// TwinCAT 3 PLC project Lynus_Standards
// Title: Lynus Standards
// Company: EfficientIO
// ProjectVersion: 1.0.0.2
// Description: Added FB BatteryInverter_11
// ProgramVersion: 3.1.4024.12
// libraries:
//   Tc2_EIB, * (Beckhoff Automation GmbH)
//   Tc2_MBus, * (Beckhoff Automation GmbH)
//   Tc2_Standard, * (Beckhoff Automation GmbH)
//   Tc2_SUPS, * (Beckhoff Automation GmbH)
//   Tc2_System, * (Beckhoff Automation GmbH)
//   Tc2_Utilities, * (Beckhoff Automation GmbH)
//   Tc3_BA_Common, * (Beckhoff Automation GmbH)
//   Tc3_JsonXml, * (Beckhoff Automation GmbH)
//   Tc3_Module, * (Beckhoff Automation GmbH)
// project tree:
//   Bussystems/DUTs intern/MBus Master/ ST_MBusMaster_KL6781_GVL.TcDUT
//   Bussystems/DUTs intern/RTU Master/ ST_MBRTUMaster_KL6xxx_GVL.TcDUT
//   Bussystems/ENUMs Internal/RTU Master/ E_MBRTUMaster_DeviceType.TcDUT, E_MBRTUMaster_ReadWriteMode.TcDUT
//   Bussystems/ENUMs/KNX Master/ E_Message_KNXMaster.TcDUT
//   Bussystems/ENUMs/MB RTU Master/ E_Message_MBRTUMaster.TcDUT
//   Bussystems/ENUMs/MBus Master/ E_Message_MBusMaster.TcDUT
//   Bussystems/FBs Internal/KNX Master/ FB_KNXMaster_Messages.TcPOU
//   Bussystems/FBs Internal/MBus Master/ FB_MBusMaster_Messages.TcPOU
//   Bussystems/FBs Internal/RTU Master/ FB_MBRTUMaster_Messages.TcPOU
//   Communicator/DUTs/ ST_BlockReadValue.TcDUT, ST_Content_Of_Document.TcDUT, ST_Infos_SubItem.TcDUT, ST_Message_In.TcDUT, ST_Message_Out.TcDUT, ST_SymbolRead.TcDUT, ST_Symbol_Info_SubItem.TcDUT, ST_Symbol_Upload_Info.TcDUT, ST_Symbol_Upload_Raw.TcDUT, ST_Var_Info.TcDUT, ST_Var_Info_EX.TcDUT, ST_Var_Info_EX_All.TcDUT, ST_Var_Info_GV.TcDUT, ST_Var_Info_ValueSend_GV.TcDUT, ST_Var_Info_ValueWrite_GV.TcDUT
//   Communicator/ENUMs/ eErrorMessage.TcDUT, eErrorReadWrite.TcDUT, eErrorVarInfo.TcDUT, eSavePositionFile.TcDUT, eSymbolTypeFromDocument.TcDUT
//   Communicator/FBs Internal/ FB_MessageRead.TcPOU, FB_MessageWrite.TcPOU, FB_ParsDocument.TcPOU, FB_VarInfo_ErrorCodes.TcPOU, FB_VarReadWrite_ErrorCodes.TcPOU
//   Energy/DUTs Internal/Battery Inverter/ ST_BatteryInverter_GVL.TcDUT
//   Energy/DUTs Internal/Battery/ ST_Battery_GVL.TcDUT
//   Energy/DUTs Internal/Beckhoff/ ST_KL3403.TcDUT
//   Energy/DUTs Internal/Electric CS/ ST_ECS_GVL.TcDUT
//   Energy/DUTs Internal/Electric Heating Element/ ST_EHE_GVL.TcDUT
//   Energy/DUTs Internal/Electric Meter/ ST_ElectricMeter_GVL.TcDUT
//   Energy/DUTs Internal/Generator/ ST_Generator_GVL.TcDUT
//   Energy/DUTs Internal/Grid/ ST_GridConnection_GVL.TcDUT
//   Energy/DUTs Internal/Heating Pump/ ST_HP_GVL.TcDUT
//   Energy/DUTs Internal/House/ ST_HouseConsumption_GVL.TcDUT
//   Energy/DUTs Internal/Other Big Consumer/ ST_OBC_GVL.TcDUT
//   Energy/DUTs Internal/PV/ ST_PV_GVL.TcDUT
//   Energy/DUTs Internal/System Time/ ST_Systemtime.TcDUT
//   Energy/DUTs Internal/Valve Control/ ST_Valve_Control_GVL.TcDUT
//   Energy/DUTs/Battery Inverter/ ST_BatteryInverter_Output.TcDUT
//   Energy/DUTs/Battery/ ST_Battery_Output.TcDUT
//   Energy/DUTs/Electric CS/ ST_ECS_Output.TcDUT, ST_Setup_ECS.TcDUT
//   Energy/DUTs/Electric Heating Element/ ST_EHE_Output.TcDUT, ST_Setup_EHE.TcDUT
//   Energy/DUTs/Electric Meter/ ST_ElectricMeter_Output_Power.TcDUT, ST_ElectricMeter_Output_Counter.TcDUT
//   Energy/DUTs/Generator/ ST_Generator_Output.TcDUT, ST_Setup_Generator.TcDUT
//   Energy/DUTs/Grid/ ST_GridConnection_Output.TcDUT
//   Energy/DUTs/Heating pump/ ST_HP_Output.TcDUT, ST_Setup_HP.TcDUT
//   Energy/DUTs/House/ ST_HouseConsumption_Output.TcDUT
//   Energy/DUTs/Other Big Consumer/ ST_OBC_Output.TcDUT, ST_Setup_OBC.TcDUT
//   Energy/DUTs/PV/ ST_PV_Output.TcDUT
//   Energy/DUTs/Temperature/ ST_InputData_KL320x.TcDUT, ST_OutputData_KL320x.TcDUT, ST_Temperature_Output.TcDUT
//   Energy/DUTs/Valve Control/ ST_Valve_Control_Output.TcDUT
//   Energy/ENUMs Internal/Temperature/ E_ChooseSensortype_KL320x.TcDUT, E_Step_Config_Terminal_KL320x.TcDUT
//   Energy/ENUMs/Battery Inverter/ E_Message_BatteryInverter.TcDUT
//   Energy/ENUMs/Battery/ E_Message_Battery.TcDUT
//   Energy/ENUMs/Electric Charging Station/ E_Message_ECS.TcDUT
//   Energy/ENUMs/Electric Heating Element/ E_Message_EHE.TcDUT
//   Energy/ENUMs/Electric Meter/ E_Message_EM.TcDUT
//   Energy/ENUMs/EMS/ E_Message_EMS.TcDUT
//   Energy/ENUMs/Generator/ E_Message_Generator.TcDUT
//   Energy/ENUMs/Grid/ E_Message_Grid.TcDUT
//   Energy/ENUMs/Heating Pump/ E_Message_HP.TcDUT
//   Energy/ENUMs/House Consumption/ E_Message_HouseC.TcDUT
//   Energy/ENUMs/Other Big Consumer/ E_Message_OBC.TcDUT
//   Energy/ENUMs/PV/ E_Message_PV.TcDUT
//   Energy/ENUMs/Temperature/ E_Message_Temperature.TcDUT
//   Energy/ENUMs/Valve Control/ E_Message_ValveControl.TcDUT
//   Energy/FBs Internal/Battery Inverter/ FB_BatteryInverter.TcPOU, FB_BatteryInverter_11.TcPOU
//   Energy/FBs Internal/Battery/ FB_Battery.TcPOU
//   Energy/FBs Internal/Beckhoff/ FB_KL3403_SimpleProcessImage.TcPOU, FB_XL1XXX_DI.TcPOU, FB_XL2XXX_DO.TcPOU, FB_XL3XXX_AI.TcPOU, FB_XL4XXX_AO.TcPOU
//   Energy/FBs Internal/Controller/ FB_PID.TcPOU
//   Energy/FBs Internal/Electric CS/ FB_ElectricChargingStation.TcPOU
//   Energy/FBs Internal/Electric Heating Element/ FB_ElectricHeatingElement.TcPOU
//   Energy/FBs Internal/Electric Meter/ FB_ElectricMeter.TcPOU
//   Energy/FBs Internal/EMS/ FB_EMS_Message.TcPOU
//   Energy/FBs Internal/Energy Counter/ FB_EnergyCounter.TcPOU
//   Energy/FBs Internal/Generator/ FB_Generator.TcPOU
//   Energy/FBs Internal/Grid/ FB_GridConnection.TcPOU
//   Energy/FBs Internal/Heating Pump/ FB_HeatingPump.TcPOU
//   Energy/FBs Internal/House/ FB_HouseConsumption.TcPOU
//   Energy/FBs Internal/Other Big Consumer/ FB_BigConsumer.TcPOU
//   Energy/FBs Internal/PV/ FB_PV_Production.TcPOU
//   Energy/FBs Internal/Valve Control/ FB_Valve_Control.TcPOU
//   General/DUTs Internal/Convert/ eByteOrder.TcDUT, ST_UN_FLOAT_CONVERT_DWORD_REAL.TcDUT, ST_UN_FLOAT_CONVERT_ULINT_LREAL.TcDUT
//   General/DUTs Internal/Devices/ ST_NumberOfDevices_GVL.TcDUT
//   General/FBs Internal/Convert/BOOL/ FB_CV_BOOL_TO_WORD.TcPOU, FB_CV_WORD_TO_BOOL.TcPOU
//   General/FBs Internal/Convert/BYTE/ FB_CV_BYTE_TO_WORD.TcPOU, FB_CV_WORD_TO_BYTE.TcPOU
//   General/FBs Internal/Convert/DINT/ FB_CV_DINT_TO_WORD.TcPOU, FB_CV_WORD_TO_DINT.TcPOU
//   General/FBs Internal/Convert/DWORD/ FB_CV_DWORD_TO_WORD.TcPOU, FB_CV_WORD_TO_DWORD.TcPOU
//   General/FBs Internal/Convert/INT/ FB_CV_INT_TO_WORD.TcPOU, FB_CV_WORD_TO_INT.TcPOU
//   General/FBs Internal/Convert/LINT/ FB_CV_LINT_TO_WORD.TcPOU, FB_CV_WORD_TO_LINT.TcPOU
//   General/FBs Internal/Convert/LREAL_FLOAT/ FB_CV_LREAL_FLOAT_TO_WORD.TcPOU, FB_CV_WORD_TO_LREAL_FLOAT.TcPOU
//   General/FBs Internal/Convert/LWORD/ FB_CV_LWORD_TO_WORD.TcPOU, FB_CV_WORD_TO_LWORD.TcPOU
//   General/FBs Internal/Convert/REAL_FLOAT/ FB_CV_REAL_FLOAT_TO_WORD.TcPOU, FB_CV_WORD_TO_REAL_FLOAT.TcPOU
//   General/FBs Internal/Convert/SINT/ FB_CV_SINT_TO_WORD.TcPOU, FB_CV_WORD_TO_SINT.TcPOU
//   General/FBs Internal/Convert/UDINT/ FB_CV_UDINT_TO_WORD.TcPOU, FB_CV_WORD_TO_UDINT.TcPOU
//   General/FBs Internal/Convert/ULINT/ FB_CV_ULINT_TO_WORD.TcPOU, FB_CV_WORD_TO_ULINT.TcPOU
//   General/FBs Internal/Convert/USINT/ FB_CV_USINT_TO_WORD.TcPOU, FB_CV_WORD_TO_USINT.TcPOU
//   General/FBs Internal/Filter/ FB_Filter.TcPOU
//   General/FBs Internal/Linear Interpolation/ FB_Lin_Interpolation.TcPOU
//   General/FBs Internal/Number Of Device/ FB_NumberOfDevice.TcPOU
//   General/FUNs Internal/ ARRAY_AVG.TcPOU, F_Scalvalue.TcPOU
//   GVL and CONST/Bussystems/ Constants_Bussystems.TcGVL, GVL_Bussystems.TcGVL
//   GVL and CONST/Energy/ Constants_Energy.TcGVL, GVL_Energy.TcGVL
//   GVL and CONST/Communicator/ GVL_Communicator.TcGVL, Constants_Communicator.TcGVL
//   GVL and CONST/General/ Constants_General.TcGVL
//   GVL and CONST/Persistent Data/ GVL_Persistent_Data.TcGVL
//   GVL and CONST/Sensors/ Constants_Sensors.TcGVL, GVL_Sensors.TcGVL
//   Persistent Data/FBs Internal/PD Slave/ FB_PersistentData_Number.TcPOU, FB_PersistentData_String.TcPOU
//   Sensors/DUTs Internal/Temperature/ ST_Temperature_GVL.TcDUT
//   Sensors/FBs Internal/Temperature/ FB_Config_KL320x.TcPOU, FB_TempSensor_M50_P200.TcPOU

// ---- Bussystems/DUTs intern/MBus Master/ST_MBusMaster_KL6781_GVL.TcDUT
{attribute 'conditionalshow'}
TYPE ST_MBusMaster_KL6781_GVL :
STRUCT
	{attribute 'hide'}
	stDataMBusCommunicationKL6781					: ST_MBus_Communication;					//Datastrcut between the KL6781 and the other Functionblocks
	{attribute 'hide'}			
	eBaudrateMBusKL6781								: E_MBus_Baudrate;							//With this Baudrate the Functionsblocks for the Counters are reading out
END_STRUCT
END_TYPE

// ---- Bussystems/DUTs intern/RTU Master/ST_MBRTUMaster_KL6xxx_GVL.TcDUT
{attribute 'conditionalshow'}
TYPE ST_MBRTUMaster_KL6xxx_GVL :
STRUCT
	{attribute 'hide'}
	bSlaveStartReadOrWrite				: BOOL;																		//RTU Slave send to the RTU Master the start for read or write command
	{attribute 'hide'}
	bTerminalIsConfigured				: BOOL;																		//The RTU Master set this Flag to True when the Terminal is successfully configured
	{attribute 'hide'}	
	bReadWriteIsDone					: BOOL;																		//The Slave Set this to True when all Registers are done. (For Eg. in the Last Step of the Statemachine) The Master Reset this Flag. So then next Modbus Adress can be processed.
	{attribute 'hide'}
	bMasterIsBusy						: BOOL;																		//RTU Master is busy. 
	{attribute 'hide'}
	bNoNewMBusAdress					: BOOL;																		//When this Flag is true, the Client Functions not can set a new Modbus Slave Adress
	{attribute 'hide'}
	byErrorWarning						: BYTE;																		//Error Warning State
	{attribute 'hide'}
	byActualMBAdressInProgrss			: BYTE;																		//Actual Modbus Slave Adress what is in Progress at the moment
	{attribute 'hide'}
	byNumberOfSlaves					: BYTE;																		//Number of Slaves on several Line
	{attribute 'hide'}
	wModbusRegister						: WORD;																		//The Modbus Register from the Slave for the Master to read/write
	{attribute 'hide'}	
	wNumberOfRegister					: WORD;																		//Number of Registers from the Slave to the Master for read/write 
	{attribute 'hide'}
	arrAllModbusSlaveAdresses			: ARRAY[1..247] OF BYTE;													//Array with all Modbuis Slave Adresses				
	{attribute 'hide'}
	arrReadOutData						: ARRAY[1..Constants_Bussystems.wQuantityOfRegistersMBRTUMaster] OF WORD;	//Data after Reading to send from the Master to the Slave
	{attribute 'hide'}
	arrWriteOutData						: ARRAY[1..Constants_Bussystems.wQuantityOfRegistersMBRTUMaster] OF WORD;	//Data to send from the Save to the Master for writing
	{attribute 'hide'}
	eMBRTUReadWriteMode					: E_MBRTUMaster_ReadWriteMode;												//Choose between the different Modbus Actions
	{attribute 'hide'}
	eMBRTUDeviceType					: E_MBRTUMaster_DeviceType;													//The Slave send to the Master the Device Type. Only the same Device Types are Allowed on 1 Backhoff Terminal
END_STRUCT
END_TYPE

// ---- Bussystems/ENUMs Internal/RTU Master/E_MBRTUMaster_DeviceType.TcDUT
{attribute 'qualified_only'}
{attribute 'strict'}
{attribute 'conditionalshow'}
TYPE E_MBRTUMaster_DeviceType :
(
	//Device Types on the RTU Bus, to configure the Terminal
	{attribute 'hide'}
	eNoModbusRTUDevice								:= 0,
	{attribute 'hide'}
	ePilotPMAC201_HW								:= 1,
	{attribute 'hide'}				
	eDrexelAWeiss_AereosilentStratosLU_Ventilation	:= 2,
	{attribute 'hide'}
	eABB_CM_UFD_M31M_NAProtection					:= 3,
	{attribute 'hide'}
	eSchrack_ECS_CIONHOME_SEMIPUBLIC				:= 4,
	{attribute 'hide'}
	ePV_DeltaSunspec								:= 5
);
END_TYPE

// ---- Bussystems/ENUMs Internal/RTU Master/E_MBRTUMaster_ReadWriteMode.TcDUT
{attribute 'qualified_only'}
{attribute 'strict'}
{attribute 'conditionalshow'}
TYPE E_MBRTUMaster_ReadWriteMode :
(
	{attribute 'hide'}
	eModbusRTUMaster_NoMode := 0,
	{attribute 'hide'}
	eModbusRTUMaster_ReadCoils	:= 1,									//Read binary Outputs
	{attribute 'hide'}
	eModbusRTUMaster_ReadInputStatus	:= 2,							//Read binary Inputs
	{attribute 'hide'}
	eModbusRTUMaster_ReadRegs	:= 3,									//Read Output Registers
	{attribute 'hide'}
	eModbusRTUMaster_ReadInputRegs	:= 4,								//Read Input Registers
	{attribute 'hide'}
	eModbusRTUMaster_WriteSingleCoil	:= 5,							//Write 1 binary Outputs
	{attribute 'hide'}
	eModbusRTUMaster_WriteSingleRegister	:= 6,						//Write a single Register
	{attribute 'hide'}
	eModbusRTUMaster_Diagnostics	:= 8,								//Send a Diagnostic request
	{attribute 'hide'}
	eModbusRTUMaster_WriteMultipleCoils	:= 15,							//Write more binary Outputs 
	{attribute 'hide'}
	eModbusRTUMaster_WriteRegs	:= 16									//Write more then one Register
);
END_TYPE

// ---- Bussystems/ENUMs/KNX Master/E_Message_KNXMaster.TcDUT
{attribute 'qualified_only'}
{attribute 'strict'}
TYPE E_Message_KNXMaster :
(
	eAllOk := 0,
	eTooMuchKNXMasters := 1,
	eNoConnectionToBackend := 2,
	eWrong_KNX_Phys_Addr := 3,
	eWrong_KNX_Group_Addr := 4,
	eWrong_KNX_Group_Len := 5,
	eWrong_KNX_No_Filter := 6,
	eWrong_KNX_Firmware := 7,
	eWrong_KNX_Mode := 8,
	eWrong_Mode := 9,
	eWrong_KNX_Firmware_B1_Necessary := 10,
	eWrong_KNX_Firmware_B3_Necessary := 11,
	eWrong_KNX_Data_Len := 12,
	eError_KNX_Service_Not_Support := 13,
	eKL6301_TP_Toggle_Error := 14,
	eTime_Out := 15,
	eKL6301_No_Response_from_Terminal := 16,
	eError_Send_8Bit_Wrong_Scaling_Mode := 17,
	eError_KNX_Phy_Addr_Not_Support := 18,
	eError_KNX_Write_Data := 19,
	eMonitor_Mode_Len_Is_Not_Ok_Must_0 := 20,
	eMonitor_Mode_Addr_Is_Not_Ok_Must_0 := 21,
	eWatchdog_Error_No_Send := 22,
	eError_KNX_No_Ack := 23,
	eError_KNX_No_Com_To_TP := 24,
	eError_TP_Temp_Warning := 25,
	eError_TP_Protocol_Error := 26,
	eError_TP_Transmitter_Error := 27,
	eError_TP_Receive_Error := 28,
	eError_TP_Slave_Collision := 29
);
END_TYPE

// ---- Bussystems/ENUMs/MB RTU Master/E_Message_MBRTUMaster.TcDUT
{attribute 'qualified_only'}
{attribute 'strict'}
TYPE E_Message_MBRTUMaster :
(
	eAllOk := 0,
	eNoTerminalConfiguration := 1,
	eTooMuchMBRTUMasters := 2,
	eNoConnectionToBackend := 3,
	eTerminalConfigurationError := 4,
	eModbusErrorIllegalFunction := 5,
	eModbusErrorIllegalDataAdress := 6,
	eModbusErrorIllegalDataValue := 7,
	eModbusErrorSlaveDeviceFailure := 8,
	eModbusErrorAcknowledge := 9,
	eModbusErrorSlaveDeviceBusy := 10,
	eModbusErrorNegativeAcknowledge := 11,
	eModbusErrorMemoryParity := 12,
	eModbusErrorGatewayPathUnavailable := 13,
	eModbusErrorGatewayTargetDeviceFailedToRespond := 14,
	eModbusErrorCharrecTimeout := 15,
	eModbusErrorIllegalDataSize := 16,
	eModbusErrorIllegalDeviceAdress := 17,
	eModbusErrorIllegalDestinationAdress := 18,
	eModbusErrorIllegalDestinationSize := 19,
	eModbusErrorNoResponse := 20,
	eModbusErrorTxBufferOverrun := 21,
	eModbusErrorSendTimeout := 22,
	eModbusErrorDataSizeOverrun := 23,
	eModbusErrorStringOverrun := 24,
	eModbusErrorInvalidPointer := 25,
	eModbusErrorCRC := 26,
	eModbusErrorInvalidMemoryAdress := 27,
	eModbusErrorTransmitBufferTooSmal := 28
);
END_TYPE

// ---- Bussystems/ENUMs/MBus Master/E_Message_MBusMaster.TcDUT
{attribute 'qualified_only'}
{attribute 'strict'}
TYPE E_Message_MBusMaster :
(
	eAllOk := 0,
	eTooMuchMBusMasters := 1,
	eNoConnectionToBackend := 2,
	eMBUSERROR_CIField_wrong_72hex_expected  := 3,
 	eMBUSERROR_no_data_received := 4,
  	eMBUSERROR_error_checksum := 5,
  	eMBUSERROR_error_in_head_data := 6,
 	eMBUSERROR_usiAddress_over_250 := 7,
  	eMBUSERROR_send_error := 8,
  	eMBUSERROR_received_address_wrong := 9,
  	eMBUSERROR_cMBUS_MaxCom_below_1 := 10,
  	eMBUSERROR_iComId_over_cMBUS_MaxCom := 11,
  	eMBUSERROR_manufacturer_sign_wrong := 12,
  	eMBUSERROR_baudrate_wrong := 13,
  	eMBUSERROR_ReceiveBufferFull := 14,
  	eMBUSERROR_E5hex_no_received := 15,
  	eMBUSERROR_no_stop_character := 16,
  	eMBUSERROR_length_wrong := 17,
  	eMBUSERROR_wrong_terminal := 18,
  	eMBUSERROR_Terminal_is_not_initialized := 19,
  	eMBUSERROR_stSecAdr_udiIdNumber_wrong := 20,
  	eMBUSERROR_missing_parts_telegram := 21,
  	eMBUSERROR_no_stop_character_received := 22,
  	eMBUSERROR_too_many_characters := 23,
  	eMBUSERROR_TimeOut_FB_KL6781 := 24,
  	eMBUSERROR_TimeOut_MeterFB := 25,
	eMBUSERROR_COM_PARAMETERCHANGED := 26,
  	eMBUSERROR_COM_TXBUFFOVERRUN := 27,
  	eMBUSERROR_COM_STRINGOVERRUN := 28,
  	eMBUSERROR_COM_ZEROCHARINVALID := 29,
  	eMBUSERROR_COM_INVALIDPOINTER := 30,
 	eMBUSERROR_COM_INVALIDRXPOINTER := 31,
  	eMBUSERROR_COM_INVALIDRXLENGTH := 32,
  	eMBUSERROR_COM_DATASIZEOVERRUN := 33,
  	eMBUSERROR_COM_INVALIDBAUDRATE := 34,
  	eMBUSERROR_COM_INVALIDNUMDATABITS := 35,
  	eMBUSERROR_COM_INVALIDNUMSTOPBITS := 36,
  	eMBUSERROR_COM_INVALIDPARITY := 37,
  	eMBUSERROR_COM_INVALIDHANDSHAKE := 38,
  	eMBUSERROR_COM_INVALIDNUMREGISTERS := 39,
  	eMBUSERROR_COM_INVALIDREGISTER := 40,
  	eMBUSERROR_COM_TIMEOUT := 41
);
END_TYPE

// ---- Communicator/DUTs/ST_BlockReadValue.TcDUT
{attribute 'conditionalshow'}
TYPE ST_BlockReadValue :
STRUCT
	{attribute 'hide'}
	udiIndexGroup			: UDINT;						//Index group from symbol  
	{attribute 'hide'}
	udiIndexOffset			: UDINT;						//Index offset from symbol
	{attribute 'hide'}
	udiLength				: UDINT;						//Index length from symbol
END_STRUCT
END_TYPE

// ---- Communicator/DUTs/ST_Content_Of_Document.TcDUT
{attribute 'conditionalshow'}
TYPE ST_Content_Of_Document :
STRUCT
	{attribute 'hide'}
	sSymbolName				: STRING(48);																				//Symbol Name
	{attribute 'hide'}
	eSymbolType				: eSymbolTypeFromDocument;																	//Symbol Type (Enum, Struct or FB)
	{attribute 'hide'}
	arrSubItemName			: ARRAY[1..Constants_Communicator.uiArraySizeOfMarkedSubItems] OF STRING(48);				//Name from the Subitems
	{attribute 'hide'}
	arrSubItemSymbolType	: ARRAY[1..Constants_Communicator.uiArraySizeOfMarkedSubItems] OF STRING(255);				//Type from the Subitems
	{attribute 'hide'}
	arrSubItemUnit			: ARRAY[1..Constants_Communicator.uiArraySizeOfMarkedSubItems] OF STRING(255);				//Unit from the SubItem
	{attribute 'hide'}
	arrSubItemTextEnum		: ARRAY[1..Constants_Communicator.uiArraySizeOfMarkedSubItems] OF STRING(48);				//Text from Enum
	{attribute 'hide'}
	arrSubItemIndexEnum		: ARRAY[1..Constants_Communicator.uiArraySizeOfMarkedSubItems] OF STRING(6);				//Index-Value from Enum
END_STRUCT
END_TYPE

// ---- Communicator/DUTs/ST_Infos_SubItem.TcDUT
{attribute 'conditionalshow'}
TYPE ST_Infos_SubItem :
STRUCT
	{attribute 'hide'}
	bIsEnum						: BOOL;						//Is true if the symbol is a enum		
	{attribute 'hide'}				
	sSubItemName				: STRING(48);				//Name of the Sub Item	
	{attribute 'hide'}								
	sSubItemType				: STRING(255);				//Type of the sub item
	{attribute 'hide'}									
	sSubItemUnit				: STRING(255);				//Unit of the sub item
	{attribute 'hide'}									
	uiSizeArray					: UINT;						//Array size if symbol type is a array
	{attribute 'hide'}
	udiSubItemGroup				: UDINT;					//Group number of sub item
	{attribute 'hide'}
	udiSubItemOffset			: UDINT;					//Offset of group number of sub item
	{attribute 'hide'}
	udiSubItemSize				: UDINT;					//Size of sub item variable in Byte 
END_STRUCT
END_TYPE

// ---- Communicator/DUTs/ST_Message_In.TcDUT
{attribute 'conditionalshow'}
TYPE ST_Message_In :
STRUCT
	{attribute 'hide'}
	sFullSymbolName				: STRING(48);															//Full Symbol name of plc variable uncoded
	{attribute 'hide'}
	sSymbolUnit					: STRING(255);															//Symbol unit of plc variable uncoded
	{attribute 'hide'}
	sSymbolType					: STRING(255);															//Symbol type of plc variable uncoded	
	{attribute 'hide'}
	arrValue					: ARRAY[1..Constants_Communicator.bySizeOfValueArray] OF STRING(30);	//Value from the Variable	
END_STRUCT
END_TYPE

// ---- Communicator/DUTs/ST_Message_Out.TcDUT
{attribute 'conditionalshow'}
TYPE ST_Message_Out :
STRUCT
	{attribute 'hide'}
	sFullSymbolName				: STRING(48);																			//Symbol name of plc variable uncoded
	{attribute 'hide'}
	sSymbolType					: STRING(255);																			//Symbol type of plc variable uncoded
	{attribute 'hide'}
	uiSizeArray					: UINT;																					//Size of actuall Array
	{attribute 'hide'}
	byReadWriteArrayNumber		: BYTE;																					//Number of the array for which the command is intended
	{attribute 'hide'}
	arrValue					: ARRAY[0..Constants_Communicator.bySizeOfReceivedValueArrayInJson] OF STRING(30);		//Value from the Variable	
END_STRUCT
END_TYPE

// ---- Communicator/DUTs/ST_SymbolRead.TcDUT
{attribute 'conditionalshow'}
TYPE ST_SymbolRead :
STRUCT
	{attribute 'hide'}
	sFullSymbolName				: STRING(48);																	//Full Symbol name of plc variable uncoded
	{attribute 'hide'}
	arrValue					: ARRAY[1..Constants_Communicator.bySizeOfValueArray] OF STRING(30);			//Value from the Variable	
END_STRUCT
END_TYPE

// ---- Communicator/DUTs/ST_Symbol_Info_SubItem.TcDUT
{attribute 'conditionalshow'}
TYPE ST_Symbol_Info_SubItem :
STRUCT
	{attribute 'hide'}
	udiSubItemGroup				: UDINT;					//Group number of sub item
	{attribute 'hide'}
	udiSubItemOffset			: UDINT;					//Offset of group number of sub item
	{attribute 'hide'}
	udiSubItemSize				: UDINT;					//Size of sub item variable in Byte
END_STRUCT
END_TYPE

// ---- Communicator/DUTs/ST_Symbol_Upload_Info.TcDUT
{attribute 'conditionalshow'}
TYPE ST_Symbol_Upload_Info :
STRUCT
	{attribute 'hide'}
	udiSymbols				: UDINT;				//Number of symbols on plc
	{attribute 'hide'}
	udiSymbolSize			: UDINT;				//Size of symbols on plc
END_STRUCT
END_TYPE

// ---- Communicator/DUTs/ST_Symbol_Upload_Raw.TcDUT
{attribute 'conditionalshow'}
TYPE ST_Symbol_Upload_Raw :
STRUCT
	{attribute 'hide'}
	udiSymbolName				: UDINT;				//Symbol name of plc variable in coded format
	{attribute 'hide'}
	udiGroup					: UDINT;				//Group number
	{attribute 'hide'}
	udiOffset					: UDINT;				//Offset of group number
	{attribute 'hide'}
	udiSize						: UDINT;				//Size of variable
	{attribute 'hide'}
	udiAdsDataType				: UDINT;				//Ads Data Type
	{attribute 'hide'}
	udiFlags					: UDINT;				//Flags
	{attribute 'hide'}
	uiNameLength				: UINT;					//Length of the symbol name
	{attribute 'hide'}
	uiTypeLength				: UINT;					//Lenght of the type in Byte it is bigdata ads type
	{attribute 'hide'}
	uiCommentLength				: UINT;					//Comment lenght
END_STRUCT
END_TYPE

// ---- Communicator/DUTs/ST_Var_Info.TcDUT
{attribute 'conditionalshow'}
TYPE ST_Var_Info :
STRUCT
	{attribute 'hide'}
	sSymbolName					: STRING(255);			//Symbol name of plc variable uncoded
	{attribute 'hide'}
	uiSizeArray					: UINT;					//Array size if symbol type is a array
	{attribute 'hide'}
	udiGroup					: UDINT;				//Group number
	{attribute 'hide'}
	udiOffset					: UDINT;				//Offset of group number
	{attribute 'hide'}
	udiSize						: UDINT;				//Size of variable
	{attribute 'hide'}
	udiFlags					: UDINT;				//Flags
	{attribute 'hide'}
	uiTypeLength				: UINT;					//Lenght of the type in Byte it is bigdata ads type
	{attribute 'hide'}
	sAdsDataType				: STRING(12);			//ADS data type	
	{attribute 'hide'}
	sSymbolType					: STRING(255);			//Symbol type of plc variable uncoded
	{attribute 'hide'}
	sSymbolComment				: STRING(255);			//Symbol comment of plc variable uncoded
END_STRUCT
END_TYPE

// ---- Communicator/DUTs/ST_Var_Info_EX.TcDUT
{attribute 'conditionalshow'}
TYPE ST_Var_Info_EX :
STRUCT
	{attribute 'hide'}
	bNoStandardDatatypeDetected	: BOOL;																					//If its true the Symbol is not a standart Data Type			
	{attribute 'hide'}
	sFullSymbolName				: STRING(48);																			//Full Symbol name of plc variable 
	{attribute 'hide'}
	sSymbolName					: STRING(255);																			//Symbol name of plc variable 
	{attribute 'hide'}
	uiSizeArray					: UINT;																					//Array size if symbol type is a array
	{attribute 'hide'}
	udiGroup					: UDINT;																				//Group number
	{attribute 'hide'}
	udiOffset					: UDINT;																				//Offset of group number
	{attribute 'hide'}
	udiSize						: UDINT;																				//Size of variable in Byte	
	{attribute 'hide'}
	uiTypeLength				: UINT;																					//Lenght of the type in Byte it is bigdata ads type
	{attribute 'hide'}
	udiFlags					: UDINT;																				//Flags
	{attribute 'hide'}
	sAdsDataType				: STRING(12);																			//ADS data type	
	{attribute 'hide'}
	sSymbolType					: STRING(255);																			//Symbol type of plc variable	
	{attribute 'hide'}
	sSymbolUnit					: STRING(255);																			//Symbol Unit
	{attribute 'hide'}
	sProjectName				: STRING(63);																			//Projekt Name			
	{attribute 'hide'}
	arrInfoSubItems				: ARRAY[1..Constants_Communicator.uiArraySizeOfMarkedSubItems] OF ST_Infos_SubItem; 	//All important infos from the SubItems it is not a standart Data Type
END_STRUCT
END_TYPE

// ---- Communicator/DUTs/ST_Var_Info_EX_All.TcDUT
{attribute 'conditionalshow'}
TYPE ST_Var_Info_EX_All :
STRUCT
	{attribute 'hide'}
	sFullSymbolName				: STRING(48);			//Full Symbol name of plc variable
	{attribute 'hide'}
	uiSizeArray					: UINT;					//Array size if symbol type is a array
	{attribute 'hide'}
	udiGroup					: UDINT;				//Group number
	{attribute 'hide'}
	udiOffset					: UDINT;				//Offset of group number
	{attribute 'hide'}
	udiSize						: UDINT;				//Size of variable in Byte	
	{attribute 'hide'}
	sSymbolType					: STRING(255);			//Symbol Type
	{attribute 'hide'}
	sSymbolUnit					: STRING(255);			//Comment from the symbol
END_STRUCT
END_TYPE

// ---- Communicator/DUTs/ST_Var_Info_GV.TcDUT
{attribute 'conditionalshow'}
TYPE ST_Var_Info_GV :
STRUCT
	{attribute 'hide'}
	sFullSymbolName				: STRING(48);			//Full Symbol name of plc variable uncoded
	{attribute 'hide'}
	uiSizeArray					: UINT;					//Array size if symbol type is a array
	{attribute 'hide'}
	udiGroup					: UDINT;				//Group number
	{attribute 'hide'}
	udiOffset					: UDINT;				//Offset of group number
	{attribute 'hide'}
	udiSize						: UDINT;				//Size of variable in Byte	
	{attribute 'hide'}
	sSymbolType					: STRING(255);			//Symbol Type
	{attribute 'hide'}
	sSymbolUnit					: STRING(255);			//Comment from the symbol	
END_STRUCT
END_TYPE

// ---- Communicator/DUTs/ST_Var_Info_ValueSend_GV.TcDUT
{attribute 'conditionalshow'}
TYPE ST_Var_Info_ValueSend_GV :
STRUCT
	//Values from ads read function
	{attribute 'hide'}
	sFullSymbolName				: STRING(48);																	//Full Symbol name of plc variable uncoded
	{attribute 'hide'}
	sSymbolType					: STRING(255);																	//Symbol type of plc variable uncoded	
	{attribute 'hide'}
	sSymbolUnit					: STRING(255);																	//Symbol Unit
	{attribute 'hide'}
	arrValue					: ARRAY[1..Constants_Communicator.bySizeOfValueArray] OF STRING(30);			//Value from the Variable
	//Values from sending function and buffer
	{attribute 'hide'}
	bBufferOK					: BOOL;																			//Buffer state ok
	{attribute 'hide'}
	bBusy						: BOOL;																			//Send Message is busy
	{attribute 'hide'}
	bErrorSending				: BOOL;																			//After send messege success a error	
	{attribute 'hide'}
	udiCountBuffer				: UDINT;																		//Return the counter of stored values in the buffer after read	
END_STRUCT
END_TYPE

// ---- Communicator/DUTs/ST_Var_Info_ValueWrite_GV.TcDUT
{attribute 'conditionalshow'}
TYPE ST_Var_Info_ValueWrite_GV :
STRUCT
	//Received from external to ads write function
	{attribute 'hide'}
	bWriteNewValue				: BOOL;																			//New Value received to write
	{attribute 'hide'}
	bSendFunctionOK				: BOOL;																			//Necessary to start read/write
	{attribute 'hide'}
	uiSizeArray					: UINT;																			//Size of actuall Array
	{attribute 'hide'}
	udiCountBuffer				: UDINT;																		//Return the counter of stored values in the reveived buffer
	{attribute 'hide'}
	sFullSymbolName				: STRING(48);																	//Full Symbol name of plc variable uncoded
	{attribute 'hide'}
	sSymbolType					: STRING(255);																	//Symbol type of plc variable uncoded	
	{attribute 'hide'}
	arrValue					: ARRAY[1..Constants_Communicator.bySizeOfValueArray] OF STRING(30);			//Value from the Variable
	//State from ads write function to received function buffer
	{attribute 'hide'}
	bBusy						: BOOL;																			//Write Message is busy
	{attribute 'hide'}
	bErrorWrite					: BOOL;																			//After write the messege success a error		
END_STRUCT
END_TYPE

// ---- Communicator/ENUMs/eErrorMessage.TcDUT
{attribute 'qualified_only'}
{attribute 'strict'}
TYPE eErrorMessage :
(
	eNoError							:= 0,
	eReceivedMessageWithError			:= 1,
	eReceivedMessageIncompatibility		:= 2,
	eCreatedMessageWithError			:= 3
);
END_TYPE

// ---- Communicator/ENUMs/eErrorReadWrite.TcDUT
{attribute 'qualified_only'}
{attribute 'strict'}
TYPE eErrorReadWrite :
(
	eNoError							:= 0,
	eErrorRead							:= 1,
	eErrorWrite							:= 2,
	eErrorSizeFloatValueRead			:= 3,
	eErrorSizeValueWrite				:= 4
);
END_TYPE

// ---- Communicator/ENUMs/eErrorVarInfo.TcDUT
{attribute 'qualified_only'}
{attribute 'strict'}
TYPE eErrorVarInfo :
(
	eNoError								:= 0,
	eArraySizeError							:= 1,
	eTimoutError							:= 2,
	eCommentLenghtError						:= 3,
	eCommentDescriptionError				:= 4,
	eSymbolTypeError						:= 5,
	eSymbolNameToLongError					:= 6,
	eReadWriteFunctionToMuch				:= 7,
	eVarInfoFunctionToMuch					:= 8,
	eSendReceiveFunctionToMuch				:= 9,
	eMoreReadWriteFuctionsAsSymbols			:= 10,
	eNoTMCFileSelected						:= 11,
	eArrayWithNoStandartDatatype			:= 12,
	eSymbolNotFoundInTMCFile				:= 13,
	eSymbolNameWithSubItemIsToLong			:= 14,
	eToMuchSubItemsInSymbol					:= 15,
	eToMuchSymbols							:= 16,
	eSubItemsInfoError						:= 17,
	eNoSendReceiveFunction					:= 18,
	eNoReadWriteFunction					:= 19,
	eNoSymbolsFound							:= 20,
	eTMCFileTimoutError						:= 100,
	eTMCFileContentOfSymbolIsToBig			:= 101,
	eTMCFileSymbolNameToLongError			:= 102,
	eTMCFileToMuchSubItemsInOneSymbol		:= 103,
	eTMCFileSubItemNameToLongError			:= 104,
	eTMCFileErrorWhenOpeningTheFile			:= 105,
	eTMCFileErrorWhenReadingTheFile			:= 106,
	eTMCFileErrorWhenClosingTheFile			:= 107,
	eTMCFileToMuchNoStandartDatatypes		:= 108,
	eTMCFileEnumNameToLongError				:= 109,
	eTMCFileEnumIndexToMuchSizes			:= 110,
	eTMCFileArraySizeError					:= 111,
	eTMCFileStringSizeError					:= 112,
	eTMCFileCheckPositionError				:= 113,
	eTMCFileSearchPositionError				:= 114,
	eTMCFileMissingSubItems					:= 115,
	eTMCFileFunctionblockAccessNotAllowed	:= 116,
	eTMCFileToMuchSubItemsInOtherSubItems	:= 117,
	eTMCFileArrayWithNoStandartDatatype		:= 118
);
END_TYPE

// ---- Communicator/ENUMs/eSavePositionFile.TcDUT
{attribute 'qualified_only'}
{attribute 'strict'}
{attribute 'conditionalshow'}
TYPE eSavePositionFile :
(
	{attribute 'hide'}
	ePostionHardDisk := 0,
	{attribute 'hide'}
	ePostionC := 1
);
END_TYPE

// ---- Communicator/ENUMs/eSymbolTypeFromDocument.TcDUT
{attribute 'qualified_only'}
{attribute 'strict'}
{attribute 'conditionalshow'}
TYPE eSymbolTypeFromDocument :
(
	{attribute 'hide'}
	eNoInformation		:= 0,
	{attribute 'hide'}
	eIsEnum				:= 1,
	{attribute 'hide'}
	eIsStruct			:= 2,
	{attribute 'hide'}
	eIsFunctionBlock	:= 3
);
END_TYPE

// ---- Energy/DUTs Internal/Battery Inverter/ST_BatteryInverter_GVL.TcDUT
{attribute 'conditionalshow'}
TYPE ST_BatteryInverter_GVL :
STRUCT
	//Data from the battery inverter to the GVL to other functions.
	{attribute 'hide'}
	bEnabled						: BOOL;							//Battery inverter enabled
	{attribute 'hide'}
	bOnOff							: BOOL;							//State from the battery inverter. On or Off
	{attribute 'hide'}
	bWorkOnIslandMode				: BOOL;							//True when the inverter work in island mode
	{attribute 'hide'}
	byErrorWarning					: BYTE;							//Show if the function has a Error or a Warning
	{attribute 'hide'}
	byPriority						: BYTE; 						//Priority of the device if controlled via the EMS block => 1 2 3 (If 0 then this device does not exist for the EMS block)	
	{attribute 'hide'}
	dwBatterySOC					: DWORD;						//The actual Battery state of Charge
	{attribute 'hide'}
	rMaxChargePower					: REAL; 						//Max. charge power battery inverter with unit kW
	{attribute 'hide'}
	rMaxDischargePower				: REAL;							//Max. discharge power battery inverter with unit kW
	{attribute 'hide'}
	lrPowerOnIslandMode				: LREAL;						//Power from the battery inverter when island mode is active with unit kW
	{attribute 'hide'}
	lrPowerNormalMode				: LREAL;						//Power from the battery inverter when normal mode is active with unit kW
	//Data from the EMS function to the GVL to the battery inverter function.
	{attribute 'hide'}
	rTargetPowerEMS					: REAL;							//Target Power -100% to +100% from the EMS function
	{attribute 'hide'}
	byReserveSOCEPO					: BYTE;							//Reserve SOC in battery for emergency power operation
	{attribute 'hide'}
	byMaxDepthOfDischargeEPO		: BYTE; 						//If islanding is active, the maximum discharge depth of the batteries can be set here until the inverter switches off.
END_STRUCT
END_TYPE

// ---- Energy/DUTs Internal/Battery/ST_Battery_GVL.TcDUT
{attribute 'conditionalshow'}
TYPE ST_Battery_GVL :
STRUCT
	//Data from the battery to the GVL to other functions.
	{attribute 'hide'}
	dwSOC								: DWORD;						//The actual Battery state of Charge
	{attribute 'hide'}
	dwSOH								: DWORD;						//The actual battery state of health
	{attribute 'hide'}
	rVoltage							: REAL;							//Battery Voltage with Unit V with max. 2 comas
	{attribute 'hide'}
	lrPower								: LREAL;						//Battery Power with unit kW
	{attribute 'hide'}
	lrPowerConsumption					: LREAL;						//Battery power consumption with unit kW (charging)
	{attribute 'hide'}
	lrPowerProduction					: LREAL;						//Battery power production with unit kW (discharging)
	{attribute 'hide'}
	lrCurrent							: LREAL;						//Battery current with unit A with max. 2 comas
	{attribute 'hide'}
	lrTemp								: LREAL;						//Battery temperarure with unit °C with max. 2 comas
	{attribute 'hide'}
	lrCapacity							: LREAL;						//Actual Battery capacity in kWh with max. 2 comas
	{attribute 'hide'}
	byErrorWarning						: BYTE;							//Show if the function has a Error or a Warning		
	{attribute 'hide'}		
	bEnabled							: BOOL;							//Battery enabled
	{attribute 'hide'}
	rMaxDcChargeCurrent					: REAL;							//Max. dc charge current battery with unit A 
	{attribute 'hide'}
	rMaxDcDischargeCurrent				: REAL;							//Max. dc discharge current battery with unit A
	{attribute 'hide'}
	rMaxChargeVoltage					: REAL;							//Max. charge voltage from the battery with unit V	
END_STRUCT
END_TYPE

// ---- Energy/DUTs Internal/Beckhoff/ST_KL3403.TcDUT
{attribute 'conditionalshow'}
TYPE ST_KL3403 :
STRUCT
	{attribute 'hide'}
	byErrorWarning				: BYTE;							//Error or Warning State
	{attribute 'hide'}
	rCurrent					: REAL;							//Current in A
	{attribute 'hide'}
	rVoltage					: REAL;							//Voltage in V
	{attribute 'hide'}
	rPower						: REAL;							//Power in W
	{attribute 'hide'}
	rPowerfactor				: REAL;							//Power factor cos phi
	{attribute 'hide'}
	rEnergy						: REAL;							//Energy in kWh
	{attribute 'hide'}
	rFrequency					: REAL;							//Frequency in Hz
	{attribute 'hide'}
	rPeakValueCurrent			: REAL;							//Peak value from the Current in A
	{attribute 'hide'}
	rPeakValueVoltage			: REAL;							//Peak value from the Voltage in V
	{attribute 'hide'}
	rPeakValuePower				: REAL;							//Peak Value from the Power in W
	{attribute 'hide'}
	rMinValueCurrent			: REAL;							//Min value from the Current in A
	{attribute 'hide'}
	rMinValueVoltage			: REAL;							//Min value from the Voltage in V
	{attribute 'hide'}
	rMinValuePower				: REAL;							//Min Value from the Power in W
END_STRUCT
END_TYPE

// ---- Energy/DUTs Internal/Electric CS/ST_ECS_GVL.TcDUT
{attribute 'conditionalshow'}
TYPE ST_ECS_GVL :
STRUCT
	//Data from the electric charging station to the GVL to other functions.
	{attribute 'hide'}
	bEnabled									: BOOL;										//Charging Station is enabled
	{attribute 'hide'}
	bIsControllable 							: BOOL;										//Charging station is controllable  
	{attribute 'hide'}
	byPriority									: BYTE; 									//Priority of the device if controlled via the EMS block => 1 2 3 (If 0 then this device does not exist for the EMS block)
	{attribute 'hide'}
	byElectricFuseLine							: BYTE; 									//Electric Fuse Line on wich the ECS is connected => 1 2 3 (If 0 then this charging station is not connected to a Electric Fuse Line)
	{attribute 'hide'}
	byErrorWarning								: BYTE;										//Show if the function has a Error or a Warning
	{attribute 'hide'}
	rMaxPower									: REAL; 									//Max. power from the charging Station with unit kW
	{attribute 'hide'}
	lrPower										: LREAL;									//Actual power charging station with unit kW
	{attribute 'hide'}
	lrPowerConsumption							: LREAL;									//Consumption charging station with unit kW
	{attribute 'hide'}
	lrPowerProduction							: LREAL;									//Production charging station with unit kW
	//Data from the EMS function to the GVL to the electric charging station function.
	{attribute 'hide'}
	rTargetPowerEMS								: REAL;										//Target power from 0% to +100% from the EMS function
END_STRUCT
END_TYPE

// ---- Energy/DUTs Internal/Electric Heating Element/ST_EHE_GVL.TcDUT
{attribute 'conditionalshow'}
TYPE ST_EHE_GVL :
STRUCT
	//Data from the electric heating element to the GVL to other functions.
	{attribute 'hide'}
	bEnabled									: BOOL;										//Heating element is enabled
	{attribute 'hide'}
	bIsStepSwitched								: BOOL;										//Heating element is step switched or not
	{attribute 'hide'}
	bIsControllable 							: BOOL;										//Heating element is controllable
	{attribute 'hide'}
	byPriority									: BYTE; 									//Priority of the device if controlled via the EMS block => 1 2 3 (If 0 then this device does not exist for the EMS block)
	{attribute 'hide'}
	byErrorWarning								: BYTE;										//Show if the function has a Error or a Warning
	{attribute 'hide'}
	byNumberOfSteps								: BYTE;										//Numer of steps form the heating element
	{attribute 'hide'}
	arrMaxPower									: ARRAY[1..10] OF REAL; 					//Maximum power of the load in kW (Per stage) (If no stage or only On Off then max power in array[1])
	{attribute 'hide'}
	lrPower										: LREAL;									//Actual power heating element with unit kW
	{attribute 'hide'}
	lrPowerConsumption							: LREAL;									//Consumption heating element with unit kW
	{attribute 'hide'}
	lrPowerProduction							: LREAL;									//Production heating element with unit kW
	//Data from the EMS function to the GVL to the electric heating element function.
	{attribute 'hide'}
	arrTargetPowerEMS							: ARRAY[1..10] OF REAL;						//Target power from 0% to +100% from the EMS function
END_STRUCT
END_TYPE

// ---- Energy/DUTs Internal/Electric Meter/ST_ElectricMeter_GVL.TcDUT
{attribute 'conditionalshow'}
TYPE ST_ElectricMeter_GVL :
STRUCT
	{attribute 'hide'}
	bEnabled									: BOOL;										//Function is enabled or not
	{attribute 'hide'}
	byErrorWarning								: BYTE;										//Show if the function has a Error or a Warning
	{attribute 'hide'}
	lrTotalCounterEnergy_Consumption			: LREAL;									//Total Counter for Energy consumption with unit kWh
	{attribute 'hide'}
	lrTotalCounterEnergy_Production				: LREAL;									//Total Counter for Energy production with unit kWh
	{attribute 'hide'}
	lrCounterEnergyT1_Consumption				: LREAL;									//Total counter for energy Tariff 1 consumption with unit kWh
	{attribute 'hide'}
	lrCounterEnergyT2_Consumption				: LREAL;									//Total counter for energy Tariff 2 consumption with unit kWh
	{attribute 'hide'}
	lrCounterEnergyT1_Production				: LREAL;									//Total counter for energy Tariff 1 production with unit kWh
	{attribute 'hide'}
	lrCounterEnergyT2_Production				: LREAL;									//Total counter for energy Tariff 2 production with unit kWh
	{attribute 'hide'}
	lrPower										: LREAL;									//Actual power with unit kW
	{attribute 'hide'}
	lrPowerConsumption							: LREAL;									//Consumption power with unit kW
	{attribute 'hide'}
	lrPowerProduction							: LREAL;									//Production power with unit kW	
END_STRUCT
END_TYPE

// ---- Energy/DUTs Internal/Generator/ST_Generator_GVL.TcDUT
{attribute 'conditionalshow'}
TYPE ST_Generator_GVL :
STRUCT
	//Generator
	{attribute 'hide'}
	bEnabled									: BOOL;									//Generator is enabled
	{attribute 'hide'}
	bOutput										: BOOL;									//Output Generator
	{attribute 'hide'}
	bSReset										: BOOL;									//Reset Generator
	{attribute 'hide'}
	byErrorWarning								: BYTE;									//Show if the function has a Error or a Warning
	{attribute 'hide'}
	lrPower										: LREAL;								//Actual power generator with unit kW
	{attribute 'hide'}
	lrPowerConsumption							: LREAL;								//Consumption generator with unit kW
	{attribute 'hide'}
	lrPowerProduction							: LREAL;								//Production generator with unit kW
END_STRUCT
END_TYPE

// ---- Energy/DUTs Internal/Grid/ST_GridConnection_GVL.TcDUT
{attribute 'conditionalshow'}
TYPE ST_GridConnection_GVL :
STRUCT
	//Grid
	{attribute 'hide'}
	bEnabled									: BOOL;							//Grid function is enabled
	{attribute 'hide'}
	byErrorWarning								: BYTE;							//Show if the function has a Error or a Warning
	{attribute 'hide'}
	lrPower										: LREAL;						//Grid power with unit kW
	{attribute 'hide'}
	lrPowerConsumption							: LREAL;						//Consumption grid with unit kW
	{attribute 'hide'}
	lrPowerProduction							: LREAL;						//Production grid with unit kW
	{attribute 'hide'}
	rSizeGridConn								: REAL;							//Size fromt the grid connection with unit kW
END_STRUCT
END_TYPE

// ---- Energy/DUTs Internal/Heating Pump/ST_HP_GVL.TcDUT
{attribute 'conditionalshow'}
TYPE ST_HP_GVL :
STRUCT
	//Data from the heating pump to the GVL to other functions.
	{attribute 'hide'}
	bEnabled									: BOOL;										//Heating pump is enabled
	{attribute 'hide'}
	bIsStepSwitched								: BOOL;										//Heating pump is step switched or not
	{attribute 'hide'}
	bIsControllable 							: BOOL;										//Heating pump is controllable
	{attribute 'hide'}
	byErrorWarning								: BYTE;										//Show if the function has a Error or a Warning
	{attribute 'hide'}
	byPriority									: BYTE; 									//Priority of the device if controlled via the EMS block => 1 2 3 (If 0 then this device does not exist for the EMS block)
	{attribute 'hide'}
	byNumberOfSteps								: BYTE;										//Numer of steps form the heating pump
	{attribute 'hide'}
	rBoilerTempHeatingSys						: REAL;										//Boiler temperature heating system
	{attribute 'hide'}
	rBoilerTempServiceWater						: REAL;										//Boiler temperature service water
	{attribute 'hide'}
	rFlowTemp									: REAL;										//Flow temperature Heat pump
	{attribute 'hide'}
	rReturnTemp									: REAL;										//Return temperature Heat pump
	{attribute 'hide'}
	rFlowTempEnergySource						: REAL;										//Flow temperature Energy Source
	{attribute 'hide'}
	rReturnTempEnergySource						: REAL;										//Return temperature Energy Source
	{attribute 'hide'}
	lrElPower									: LREAL;									//Electric Power Heating pump with unit kW
	{attribute 'hide'}
	lrElPowerConsumption						: LREAL;									//Consumption heating pump with unit kW
	{attribute 'hide'}
	lrElPowerProduction							: LREAL;									//Production heating pump with unit kW
	{attribute 'hide'}
	arrMaxPower									: ARRAY[1..2] OF REAL; 						//Maximum power of the load in kW (Per stage) (If no stage or only On Off then max power in array[1])
	//Data from the EMS function to the GVL to the heating pump function.
	{attribute 'hide'}
	bExternalOnCommand							: BOOL;										//Use to switch on the HP in lower tariff when we have not enough surplues power in the next 24 Hours.
	{attribute 'hide'}
	arrTargetPowerEMS							: ARRAY[1..2] OF REAL;						//Target power from 0% to +100% from the EMS function
END_STRUCT
END_TYPE

// ---- Energy/DUTs Internal/House/ST_HouseConsumption_GVL.TcDUT
{attribute 'conditionalshow'}
TYPE ST_HouseConsumption_GVL :
STRUCT
	//House Consumption
	{attribute 'hide'}
	bEnabled									: BOOL;								//House consumption function enabled
	{attribute 'hide'}
	byErrorWarning								: BYTE;								//Show if the function has a Error or a Warning
	{attribute 'hide'}
	lrPower										: LREAL;							//House consumption with unit kW
	{attribute 'hide'}
	lrPowerConsumption							: LREAL;							//Consumption House consumption with unit kW
	{attribute 'hide'}
	lrPowerProduction							: LREAL;							//Production House consumption with unit kW
END_STRUCT
END_TYPE

// ---- Energy/DUTs Internal/Other Big Consumer/ST_OBC_GVL.TcDUT
{attribute 'conditionalshow'}
TYPE ST_OBC_GVL :
STRUCT
	//Data from the big consumer to the GVL to other functions.
	{attribute 'hide'}
	bEnabled									: BOOL;										//Big consumer is enabled
	{attribute 'hide'}
	bIsControllable 							: BOOL;										//Big Consumer is controllable  
	{attribute 'hide'}
	byErrorWarning								: BYTE;										//Show if the function has a Error or a Warning
	{attribute 'hide'}
	byPriority									: BYTE; 									//Priority of the device if controlled via the EMS block => 1 2 3 (If 0 then this device does not exist for the EMS block)
	{attribute 'hide'}
	lrPower										: LREAL;									//Actual power big consumer with unit kW
	{attribute 'hide'}
	lrPowerConsumption							: LREAL;									//Consumption big consumer with unit kW
	{attribute 'hide'}
	lrPowerProduction							: LREAL;									//Production big consumer with unit kW
	{attribute 'hide'}
	rMaxPower									: REAL; 									//Max. power from the big consumer with unit kW
	//Data from the EMS function to the GVL to the big consumer function.
	{attribute 'hide'}
	rTargetPowerEMS								: REAL;										//Target power from 0% to +100% from the EMS function
END_STRUCT
END_TYPE

// ---- Energy/DUTs Internal/PV/ST_PV_GVL.TcDUT
{attribute 'conditionalshow'}
TYPE ST_PV_GVL :
STRUCT
	//PV
	{attribute 'hide'}
	bEnabled									: BOOL;							//Pv function is enabled
	{attribute 'hide'}
	byErrorWarning								: BYTE;							//Show if the function has a Error or a Warning
	{attribute 'hide'}
	lrPower										: LREAL;						//Pv power with unit kW
	{attribute 'hide'}
	lrPowerConsumption							: LREAL;						//Consumption pv with unit kW
	{attribute 'hide'}
	lrPowerProduction							: LREAL;						//Production pv with unit kW
END_STRUCT
END_TYPE

// ---- Energy/DUTs Internal/System Time/ST_Systemtime.TcDUT
{attribute 'conditionalshow'}
TYPE ST_Systemtime :
STRUCT
	{attribute 'hide'}
	wHour				: WORD;						//Hour from the windows system time
	{attribute 'hide'}
	wMinute				: WORD;						//Minute from the windows system time
	{attribute 'hide'}
	wSecond				: WORD;						//Second from the windows system time
	{attribute 'hide'}
	wMilisecond			: WORD;						//Millisecond from the windows system time
	{attribute 'hide'}
	wDay				: WORD;						//Day from the windows system time
	{attribute 'hide'}
	wMonth				: WORD;						//Month from the windows system time
	{attribute 'hide'}
	wYear				: WORD;						//Year from the windows system time
	{attribute 'hide'}
	wWeekday			: WORD;						//Weekday from the windows system time (0..6) (0=> Sunday 1-6 => Monday..Saturday)
END_STRUCT
END_TYPE

// ---- Energy/DUTs Internal/Valve Control/ST_Valve_Control_GVL.TcDUT
{attribute 'conditionalshow'}
TYPE ST_Valve_Control_GVL :
STRUCT
	{attribute 'hide'}
	bEnabled						: BOOL;							//Valve control function is enabled
	{attribute 'hide'}
	bValvePos						: BOOL;							//Actual Valve Position
	{attribute 'hide'}
	byErrorWarning					: BYTE;							//Show if the function has a Error or a Warning
END_STRUCT
END_TYPE

// ---- Energy/DUTs/Battery Inverter/ST_BatteryInverter_Output.TcDUT
TYPE ST_BatteryInverter_Output :
STRUCT
	bEnabled						: BOOL;							//{#lynus.ag#()} //Battery inverter enabled
	bOnOff							: BOOL;							//State from the battery inverter. On or Off
	bWorkOnIslandMode				: BOOL;							//True when the inverter work in island mode
	bStateReset						: BOOL;							//{#lynus.ag#()} //State of the Reset
	byErrorWarning					: BYTE;							//Show if the function has a Error or a Warning
	byPriority						: BYTE; 						//Priority of the device if controlled via the EMS block = 1 2 3 (If 0 then this device does not exist for the EMS block)	
	rTargetPower					: REAL;							//{#lynus.ag#()} //Target Power from -100% to +100%
	rMaxChargePower					: REAL; 						//Max. charge power battery inverter with unit kW
	rMaxDischargePower				: REAL;							//Max. discharge power battery inverter with unit kW
	lrPowerNormalMode				: LREAL;						//Power from the battery inverter when normal mode is active with unit kW
	lrPowerOnIslandMode				: LREAL;						//Power from the battery inverter when island mode is active with unit kW
	eMessage						: E_Message_BatteryInverter;	//Message from the Battery inverter
END_STRUCT
END_TYPE

// ---- Energy/DUTs/Battery/ST_Battery_Output.TcDUT
TYPE ST_Battery_Output :
STRUCT
	bEnabled									: BOOL;							//Battery enabled
	byErrorWarning								: BYTE;							//Show if the function has a Error or a Warning		
	dwSOC										: DWORD;						//{#lynus.ag#()} //The actual Battery state of Charge
	dwSOH										: DWORD;						//The actual battery state of health
	rBatteryVoltage								: REAL;							//Battery Voltage with Unit V with max. 2 comas
	rMaxDcChargeCurrent							: REAL;							//Max. dc charge current battery with unit A 
	rMaxDcDischargeCurrent						: REAL;							//Max. dc discharge current battery with unit A
	rMaxChargeVoltage							: REAL;							//Max. charge voltage from the battery with unit V	
	lrPower										: LREAL;						//{#lynus.ag#()} //Battery Power with unit kW
	lrPowerConsumption							: LREAL;						//Battery power consumption with unit kW (charging)
	lrPowerProduction							: LREAL;						//Battery power production with unit kW (discharging)
	lrCurrent									: LREAL;						//Battery current with unit A with max. 2 comas
	lrTemp										: LREAL;						//Battery temperarure with unit °C with max. 2 comas
	lrCapacity									: LREAL;						//{#lynus.ag#()} //Actual Battery capacity in kWh with max. 2 comas	
	eMessage									: E_Message_Battery;			//Message from the Battery				
END_STRUCT
END_TYPE

// ---- Energy/DUTs/Electric CS/ST_ECS_Output.TcDUT
TYPE ST_ECS_Output :
STRUCT
	bOutput										: BOOL;										//Output charging station = Target power > 0
	bOutputOnOff								: BOOL;										//Output charging station = Target power >= 100
	bEnabled									: BOOL;										//{#lynus.ag#()} //Charging Station is enabled
	bCarConnected								: BOOL;										//Car is connected with the charging station
	bSOnEmergPowerOff							: BOOL;										//Shows the state of the bOnEmergPowerOff input from the setups
	bSManualyOn									: BOOL;										//Shows the state of the bManualyOn input from the setups
	byPriority									: BYTE; 									//Priority of the device if controlled via the EMS block = 1 2 3 (If 0 then this device does not exist for the EMS block)
	bySManualyTargetPower						: BYTE;										//Shows the state of the byManualyTargetPower input from the setups
	bySCSMinPower								: BYTE;										//{#lynus.ag#()} //Shows the state of the bySCMinPower input from the setups
	byErrorWarning								: BYTE;										//Show if the function has a Error or a Warning
	rMaxPower									: REAL; 									//Max. power from the charging Station with unit kW
	rTargetPower								: REAL;										//{#lynus.ag#()} //Target power from 0% to +100%
	rTargetChargeCurrent						: REAL;										//Target charge current for charging station with unit A
	lrTotalCounterEnergy_Consumption			: LREAL;									//Total Counter for Energy consumption with unit kWh
	lrTotalCounterEnergy_Production				: LREAL;									//Total Counter for Energy production with unit kWh
	lrCounterEnergyT1_Consumption				: LREAL;									//Total counter for energy Tariff 1 consumption with unit kWh
	lrCounterEnergyT2_Consumption				: LREAL;									//Total counter for energy Tariff 2 consumption with unit kWh
	lrCounterEnergyT1_Production				: LREAL;									//Total counter for energy Tariff 1 production with unit kWh
	lrCounterEnergyT2_Production				: LREAL;									//Total counter for energy Tariff 2 production with unit kWh
	lrTotalPower								: LREAL;									//Actual total power charging station with unit kW
	lrTotalPowerConsumption						: LREAL;									//Consumption total charging station with unit kW
	lrTotalPowerProduction						: LREAL;									//Production total charging station with unit kW
	arrSocketStateECS							: ARRAY[1..4] OF WORD;						//Show the State from each socket of the Electric Charging station. (0= No information, 1= ECS is Free, 2= Car Connected, 3 = Car is charging)
	arrSocketSOCCar								: ARRAY[1..4] OF DWORD;						//Actual SOC from the car of each socket
	arrChargingTimeInMin						: ARRAY[1..4] OF REAL;						//Charging time from the car in minutes from each socket
	arrSocketEnergySession						: ARRAY[1..4] OF LREAL;;					//Energy in kWh from the actual Session
	arrSocketPower								: ARRAY[1..4] OF LREAL;;					//Power in kW from each socket
	eMessage									: E_Message_ECS;							//Message from the ECS
END_STRUCT
END_TYPE

// ---- Energy/DUTs/Electric CS/ST_Setup_ECS.TcDUT
TYPE ST_Setup_ECS :
STRUCT
	bOnEmergPowerOff				: BOOL;				//When emergency power is active then user can choose if the device is on or switch automatic off
	bManualyOn						: BOOL;				//Switch the device manualy on
	byPriority						: BYTE; 			//{#lynus.ag#()} //Priority of the device if controlled via the EMS block = 1 2 3 (If 0 then this device does not exist for the EMS block)
	byEnableSOC						: BYTE; 			//{#lynus.ag#()} //Enable the device when the battery SOC is greater than equal this value
	byDisableSOC					: BYTE; 			//{#lynus.ag#()} //Disable the device when the battery SOC is smaler than equal this value
	byManualyTargetPower			: BYTE;				//% of the max Power in kW when the Device is manually on
	byCSMinPower					: BYTE;				//{#lynus.ag#()} //Min power in % of the max power in kW. The charging station is operated with this power even if there is no surplus.
	rMaxPower						: REAL; 			//{#lynus.ag#()} //Max. power from the charging Station with unit kW
END_STRUCT
END_TYPE

// ---- Energy/DUTs/Electric Heating Element/ST_EHE_Output.TcDUT
TYPE ST_EHE_Output :
STRUCT
	bOutput										: BOOL;										//Output heating element = Target power > 0
	bOutputOnOff								: BOOL;										//Output heating element = Target power >= 100
	bEnabled									: BOOL;										//{#lynus.ag#()} //Heating element is enabled
	bIsStepSwitched								: BOOL;										//Heating element is step switched or not
	bSOnEmergPowerOff							: BOOL;										//Shows the state of the bOnEmergPowerOff input from the setups
	bSManualyOn									: BOOL;										//Shows the state of the bManualyOn input from the setups
	bSTimeEnabled								: BOOL;										//{#lynus.ag#()} //Shows the state of the bTimeEnabled input from the setups
	bSDisableLegionellaPr						: BOOL;										//Shows the state of the bDisableLegionellaProtection input from the setups
	byNumberOfSteps								: BYTE;										//Numer of steps form the heating element
	byPriority									: BYTE; 									//Priority of the device if controlled via the EMS block = 1 2 3 (If 0 then this device does not exist for the EMS block)
	bySManualyTargetPower						: BYTE;										//Shows the state of the byManualyTargetPower input from the setups
	byErrorWarning								: BYTE;										//Show if the function has a Error or a Warning
	rTempInBoiler								: REAL;										//{#lynus.ag#()} //Temperature in the boiler which is heated with the heating element
	arrMaxPower									: ARRAY[1..10] OF REAL; 					//Maximum power of the load in kW (Per stage) (If no stage or only On Off then max power in array[1])
	rTargetPower								: REAL;										//{#lynus.ag#()} //Target power from 0% to +100%
	lrTotalCounterEnergy_Consumption			: LREAL;									//Total Counter for Energy consumption with unit kWh
	lrTotalCounterEnergy_Production				: LREAL;									//Total Counter for Energy production with unit kWh
	lrCounterEnergyT1_Consumption				: LREAL;									//Total counter for energy Tariff 1 consumption with unit kWh
	lrCounterEnergyT2_Consumption				: LREAL;									//Total counter for energy Tariff 2 consumption with unit kWh
	lrCounterEnergyT1_Production				: LREAL;									//Total counter for energy Tariff 1 production with unit kWh
	lrCounterEnergyT2_Production				: LREAL;									//Total counter for energy Tariff 2 production with unit kWh
	lrPower										: LREAL;									//Actual power from the heating element with unit kW
	lrPowerConsumption							: LREAL;									//Consumption from the heating element with unit kW
	lrPowerProduction							: LREAL;									//Production from the heating element with unit kW
	eMessage									: E_Message_EHE;							//Message from the EHE
END_STRUCT
END_TYPE

// ---- Energy/DUTs/Electric Heating Element/ST_Setup_EHE.TcDUT
TYPE ST_Setup_EHE :
STRUCT
	bOnEmergPowerOff				: BOOL;			//When emergency power is active then user can choose if the device is on or switch automatic off
	bTimeEnabled					: BOOL;			//{#lynus.ag#()} //Heating element enabled only between the specified time if the temperature falls below the on temperature.
	bDisableLegionellaPr			: BOOL;			//Here the legionella protection can be deactivated. This is useful if the boiler has legionella protection by itself.
	bManualyOn						: BOOL;			//Switch the device manualy on
	byManualyTargetPower			: BYTE;			//% of the max Power in kW when the Device is manually on
	byPriority						: BYTE; 		//{#lynus.ag#()} //Priority of the device if controlled via the EMS block = 1 2 3 (If 0 then this device does not exist for the EMS block)
	byEnableSOC						: BYTE; 		//{#lynus.ag#()} //Enable the device when the battery SOC is greater than equal this value
	byDisableSOC					: BYTE; 		//{#lynus.ag#()} //Disable the device when the battery SOC is smaler than equal this value
	byHourOn						: BYTE;			//{#lynus.ag#()} //Hour from which the heating element can switch on
	byMinutesOn						: BYTE;			//{#lynus.ag#()} //Minutes from which the heating element can switch on
	byHourOff						: BYTE;			//{#lynus.ag#()} //Hour from which the heating element can switch off
	byMinutesOff					: BYTE;			//{#lynus.ag#()} //Minutes from which the heating element can switch off
	uiTargetTempOn					: UINT;			//{#lynus.ag#()} //Below this temperature value, the heating element is switched on in normal mode.
	uiTargetTempOff					: UINT; 		//{#lynus.ag#()} //When the temperature reaches this value in normal operation, the heating element switches off.
	uiTargetTempMax					: UINT;			//{#lynus.ag#()} //Temperature setpoint that is approached in the event of excess power.(Overheating)
	rMaxPower1						: REAL;			//{#lynus.ag#()} //Maximum power of the load in kW (1 Step) (If the Deice is not step switched or only On Off then enter only here the max power 1 time)
	rMaxPower2						: REAL;			//{#lynus.ag#()} //Maximum power of the load in kW (2 Step)
	rMaxPower3						: REAL;			//{#lynus.ag#()} //Maximum power of the load in kW (3 Step)
	rMaxPower4						: REAL;			//{#lynus.ag#()} //Maximum power of the load in kW (4 Step)
	rMaxPower5						: REAL;			//{#lynus.ag#()} //Maximum power of the load in kW (5 Step)
	rMaxPower6						: REAL;			//{#lynus.ag#()} //Maximum power of the load in kW (6 Step)
	rMaxPower7						: REAL;			//{#lynus.ag#()} //Maximum power of the load in kW (7 Step)
	rMaxPower8						: REAL;			//{#lynus.ag#()} //Maximum power of the load in kW (8 Step)
	rMaxPower9						: REAL;			//{#lynus.ag#()} //Maximum power of the load in kW (9 Step)
	rMaxPower10						: REAL;			//{#lynus.ag#()} //Maximum power of the load in kW (10 Step)
END_STRUCT
END_TYPE

// ---- Energy/DUTs/Electric Meter/ST_ElectricMeter_Output_Power.TcDUT
TYPE ST_ElectricMeter_Output_Power :
STRUCT
	bEnabled									: BOOL;										//Electric Meter is enabled or not
	byErrorWarning								: BYTE;										//Show if the function has a Error or a Warning
	lrPowerTotal								: LREAL;									//Actual power with unit kW
	lrPowerConsumption							: LREAL;									//Consumption with unit kW
	lrPowerProduction							: LREAL;									//Production with unit kW
	lrReactivePowerTotal						: LREAL;									//Reactive Power with unit kvar
	lrApparentPowerTotal						: LREAL;									//Apparent Power with unit KVA	
	lrFrequency									: LREAL;									//Frequency with unit HZ
	lrVoltageL1N								: LREAL;									//Voltage L1 to N with unit V 
	lrVoltageL1L2								: LREAL;									//Voltage L1 to L2 with unit V
	lrCurrentL1									: LREAL;									//Current L1 with unit A
	lrPowerL1									: LREAL;									//Power L1 with unit KW
	lrVoltageL2N								: LREAL;									//Voltage L2 to N with unit V
	lrVoltageL2L3								: LREAL;									//Voltage L1 to L3 with unit V
	lrCurrentL2									: LREAL;									//Current L2 winth unit A
	lrPowerL2									: LREAL;									//Power L2 with unit kW
	lrVoltageL3N								: LREAL;									//Voltage L3 to N with unit V
	lrVoltageL3L1								: LREAL;									//Voltage L3 to L1 with unit V
	lrCurrentL3									: LREAL;									//Current L3 with unit A
	lrPowerL3									: LREAL;									//Power L3 with unit kW	
	eMessage									: E_Message_EM;								//Message from the EM			
END_STRUCT
END_TYPE

// ---- Energy/DUTs/Electric Meter/ST_ElectricMeter_Output_Counter.TcDUT
TYPE ST_ElectricMeter_Output_Counter :
STRUCT
	lrTotalCounterEnergy_Production				: LREAL;									//Total Counter for Energy production with unit kWh
	lrTotalCounterEnergy_Consumption			: LREAL;									//Total Counter for Energy consumption with unit kWh
	lrCounterEnergyT1_Consumption				: LREAL;									//Total counter for energy Tariff 1 consumption with unit kWh
	lrCounterEnergyT2_Consumption				: LREAL;									//Total counter for energy Tariff 2 consumption with unit kWh
	lrCounterEnergyT1_Production				: LREAL;									//Total counter for energy Tariff 1 production with unit kWh
	lrCounterEnergyT2_Production				: LREAL;									//Total counter for energy Tariff 2 production with unit kWh
END_STRUCT
END_TYPE

// ---- Energy/DUTs/Generator/ST_Generator_Output.TcDUT
TYPE ST_Generator_Output :
STRUCT
	bEnabled									: BOOL;									//{#lynus.ag#()} //Generator is enabled
	bOutput										: BOOL;									//Output Generator
	bSReset										: BOOL;									//{#lynus.ag#()} //Reset Generator
	byErrorWarning								: BYTE;									//Show if the function has a Error or a Warning
	lrPower										: LREAL;								//Actual power generator with unit kw
	lrPowerConsumption							: LREAL;								//Consumption generator with unit kW
	lrPowerProduction							: LREAL;								//Production generator with unit kW
	lrTotalCounterEnergy_Consumption			: LREAL;								//Total Counter for Energy consumption with unit kWh
	lrTotalCounterEnergy_Production				: LREAL;								//Total Counter for Energy production with unit kWh
	lrCounterEnergyT1_Consumption				: LREAL;								//Total counter for energy Tariff 1 consumption with unit kWh
	lrCounterEnergyT2_Consumption				: LREAL;								//Total counter for energy Tariff 2 consumption with unit kWh
	lrCounterEnergyT1_Production				: LREAL;								//Total counter for energy Tariff 1 production with unit kWh
	lrCounterEnergyT2_Production				: LREAL;								//Total counter for energy Tariff 2 production with unit kWh
	eMessage									: E_Message_Generator;					//Message from the Generator
END_STRUCT
END_TYPE

// ---- Energy/DUTs/Generator/ST_Setup_Generator.TcDUT
TYPE ST_Setup_Generator :
STRUCT
	bReset						: BOOL;								//{#lynus.ag#()} //Resets an existing error on the generators, only then the generator can restart again.
	byEnableSOC					: BYTE; 							//{#lynus.ag#()} //When battery SOC falling below this value the generator is switched on
	byDisableSOC				: BYTE; 							//{#lynus.ag#()} //When battery SOC this value is exceeded, the generator is switched on
END_STRUCT
END_TYPE

// ---- Energy/DUTs/Grid/ST_GridConnection_Output.TcDUT
TYPE ST_GridConnection_Output :
STRUCT
	byErrorWarning								: BYTE;									//Show if the function has a Error or a Warning
	bEnabled									: BOOL;									//Grid function is enabled
	lrTotalCounterEnergy_Consumption			: LREAL;								//Total Counter for Energy consumption with unit kWh
	lrTotalCounterEnergy_Production				: LREAL;								//Total Counter for Energy production with unit kWh
	lrCounterEnergyT1_Consumption				: LREAL;								//Total counter for energy Tariff 1 consumption with unit kWh
	lrCounterEnergyT2_Consumption				: LREAL;								//Total counter for energy Tariff 2 consumption with unit kWh
	lrCounterEnergyT1_Production				: LREAL;								//Total counter for energy Tariff 1 production with unit kWh
	lrCounterEnergyT2_Production				: LREAL;								//Total counter for energy Tariff 2 production with unit kWh
	lrPower										: LREAL;								//{#lynus.ag#()} //Actual power from the grid with unit kW
	lrPowerConsumption							: LREAL;								//Consumption grid with unit kW
	lrPowerProduction							: LREAL;								//Production grid with unit kW
	rSizeGridConn								: REAL;									//Max size from the grid connection with unit KW
	eMessage									: E_Message_Grid;						//Message from the Grid
END_STRUCT
END_TYPE

// ---- Energy/DUTs/Heating pump/ST_HP_Output.TcDUT
TYPE ST_HP_Output :
STRUCT
	bOutput										: BOOL;										//Output heating Pump
	bEnabled									: BOOL;										//{#lynus.ag#()} //Heating pump is enabled
	bSReset										: BOOL;										//{#lynus.ag#()} //Reset heating pump
	bIsStepSwitched								: BOOL;										//Heating pump is step switched or not
	bSOnEmergPowerOff							: BOOL;										//Shows the state of the bOnEmergPowerOff input from the setups
	bSManualyOn									: BOOL;										//Shows the state of the bManualyOn input from the setups
	bSTimeEnabled								: BOOL;										//{#lynus.ag#()} //Shows the state of the bTimeEnabled input from the setups
	bExtOnCommandIsActive						: BOOL;										//Shows that the pump runs at the moment with the external on command
	byErrorWarning								: BYTE;										//Show if the function has a Error or a Warning
	byNumberOfSteps								: BYTE;										//Numer of steps form the heating pump
	byPriority									: BYTE; 									//Priority of the device if controlled via the EMS block = 1 2 3 (If 0 then this device does not exist for the EMS block)
	bySManualyTargetPower						: BYTE;										//Shows the state of the byManualyTargetPower input from the setups
	bySTimeEnabledTargetPower					: BYTE;										//{#lynus.ag#()} //Shows the state of the byTimeEnabledTargetPower input from the setups
	rBoilerTempHeatingSys						: REAL;										//Boiler temperature heating system
	rBoilerTempServiceWater						: REAL;										//Boiler temperature service water
	rFlowTemp									: REAL;										//Flow temperature Heat pump
	rReturnTemp									: REAL;										//Return temperature Heat pump
	rFlowTempEnergySource						: REAL;										//Flow temperature Energy Source
	rReturnTempEnergySource						: REAL;										//Return temperature Energy Source
	arrMaxPower									: ARRAY[1..2] OF REAL; 						//Maximum power of the load in kW (Per stage) (If no stage or only On Off then max power in array[1])
	rTargetPower								: REAL;										//{#lynus.ag#()} //Target power from 0% to +100%
	lrElPower									: LREAL;									//Electric Power Heating pump with unit kW
	lrElPowerConsumption						: LREAL;									//Consumption heating pump with unit kW
	lrElPowerProduction							: LREAL;									//Production heating pump with unit kW
	lrTotalCounterEnergy_Consumption			: LREAL;									//Total Counter for Energy consumption with unit kWh
	lrTotalCounterEnergy_Production				: LREAL;									//Total Counter for Energy production with unit kWh
	lrCounterEnergyT1_Consumption				: LREAL;									//Total counter for energy Tariff 1 consumption with unit kWh
	lrCounterEnergyT2_Consumption				: LREAL;									//Total counter for energy Tariff 2 consumption with unit kWh
	lrCounterEnergyT1_Production				: LREAL;									//Total counter for energy Tariff 1 production with unit kWh
	lrCounterEnergyT2_Production				: LREAL;									//Total counter for energy Tariff 2 production with unit kWh
	lrCounterThermalHeatingSys					: LREAL;									//Total meter reading thermal for heating in kwh
	lrCounterThermalServiceWater				: LREAL;									//Total meter reading thermal for the domestic water in kwh
	eMessage									: E_Message_HP;								//Message from the HP
END_STRUCT
END_TYPE

// ---- Energy/DUTs/Heating pump/ST_Setup_HP.TcDUT
TYPE ST_Setup_HP :
STRUCT
	bOnEmergPowerOff				: BOOL;								//When emergency power is active then user can choose if the device is on or switch automatic off
	bTimeEnabled					: BOOL;								//{#lynus.ag#()} //If True, the heat pump will be switched to the elevated mode between the specified time
	bReset							: BOOL;								//{#lynus.ag#()} //Resets the error or the warning of the heat pump internally in the FB and if necessary externally if present.
	bManualyOn						: BOOL;								//Switch the device manualy on
	byManualyTargetPower			: BYTE;								//% of the max Power in kW when the Device is manually on
	byPriority						: BYTE; 							//{#lynus.ag#()} //Priority of the device if controlled via the EMS block = 1 2 3 (If 0 then this device does not exist for the EMS block)
	byEnableSOC						: BYTE; 							//{#lynus.ag#()} //Enable the device when the battery SOC is greater than equal this value
	byDisableSOC					: BYTE; 							//{#lynus.ag#()} //Disable the device when the battery SOC is smaler than equal this value 
	byTimeEnabledTargetPower		: BYTE;								//{#lynus.ag#()} //% power to the output within release time, if the heat pump is not step switched
	byHourOn						: BYTE;								//{#lynus.ag#()} //Hour from which the heating pump can work in increased operation 
	byMinutesOn						: BYTE;								//{#lynus.ag#()} //Minutes from which the heating pump can work in increased operation
	byHourOff						: BYTE;								//{#lynus.ag#()} //Hour from which the heating pump can't work in increased operation 
	byMinutesOff					: BYTE;								//{#lynus.ag#()} //Minutes from which the heating pump can't work in increased operation
	rMaxPower1						: REAL;								//{#lynus.ag#()} //Maximum power of the load in kW (1 Step) 1 = Increased operation 
	rMaxPower2						: REAL;								//{#lynus.ag#()} //Maximum power of the load in kW (2 Step) 2 = Maximum operation
END_STRUCT
END_TYPE

// ---- Energy/DUTs/House/ST_HouseConsumption_Output.TcDUT
TYPE ST_HouseConsumption_Output :
STRUCT
	bEnabled									: BOOL;									//{#lynus.ag#()} //House consumption function enabled
	byErrorWarning								: BYTE;									//Show if the function has a Error or a Warning
	lrTotalCounterEnergy_Consumption			: LREAL;								//Total Counter for Energy consumption with unit kWh
	lrTotalCounterEnergy_Production				: LREAL;								//Total Counter for Energy production with unit kWh
	lrCounterEnergyT1_Consumption				: LREAL;								//Total counter for energy Tariff 1 consumption with unit kWh
	lrCounterEnergyT2_Consumption				: LREAL;								//Total counter for energy Tariff 2 consumption with unit kWh
	lrCounterEnergyT1_Production				: LREAL;								//Total counter for energy Tariff 1 production with unit kWh
	lrCounterEnergyT2_Production				: LREAL;								//Total counter for energy Tariff 2 production with unit kWh
	lrPower										: LREAL;								//House consumption with unit kW
	lrPowerConsumption							: LREAL;								//Consumption House consumption with unit kW
	lrPowerProduction							: LREAL;								//Production House consumption with unit kW
	eMessage									: E_Message_HouseC;						//Message from the House consumption
END_STRUCT
END_TYPE

// ---- Energy/DUTs/Other Big Consumer/ST_OBC_Output.TcDUT
TYPE ST_OBC_Output :
STRUCT
	bOutput										: BOOL;										//Output big consumer = Target power > 0
	bOutputOnOff								: BOOL;										//Output big consumer = Target power >= 100
	bEnabled									: BOOL;										//{#lynus.ag#()} //Big consumer is enabled
	bSOnEmergPowerOff							: BOOL;										//Shows the state of the bOnEmergPowerOff input from the setups
	bSManualyOn									: BOOL;										//Shows the state of the bManualyOn input from the setups
	byPriority									: BYTE; 									//Priority of the device if controlled via the EMS block = 1 2 3 (If 0 then this device does not exist for the EMS block)
	byErrorWarning								: BYTE;										//Show if the function has a Error or a Warning
	bySManualyTargetPower						: BYTE;										//Shows the state of the byManualyTargetPower input from the setups
	rMaxPower									: REAL; 									//Max. power from the big consumer with unit kW
	rTargetPower								: REAL;										//{#lynus.ag#()} //Target power from 0% to +100%
	lrTotalCounterEnergy_Consumption			: LREAL;									//Total Counter for Energy consumption with unit kWh
	lrTotalCounterEnergy_Production				: LREAL;									//Total Counter for Energy production with unit kWh
	lrCounterEnergyT1_Consumption				: LREAL;									//Total counter for energy Tariff 1 consumption with unit kWh
	lrCounterEnergyT2_Consumption				: LREAL;									//Total counter for energy Tariff 2 consumption with unit kWh
	lrCounterEnergyT1_Production				: LREAL;									//Total counter for energy Tariff 1 production with unit kWh
	lrCounterEnergyT2_Production				: LREAL;									//Total counter for energy Tariff 2 production with unit kWh
	lrPower										: LREAL;									//Actual power big consumer with unit kW
	lrPowerConsumption							: LREAL;									//Consumption big consumer with unit kW
	lrPowerProduction							: LREAL;									//Production big consumer with unit kW
	eMessage									: E_Message_OBC;							//Message from the OBC
END_STRUCT
END_TYPE

// ---- Energy/DUTs/Other Big Consumer/ST_Setup_OBC.TcDUT
TYPE ST_Setup_OBC :
STRUCT
	bOnEmergPowerOff				: BOOL;										//When emergency power is active then user can choose if the device is on or switch automatic off
	bManualyOn						: BOOL;										//Switch the device manualy on
	byManualyTargetPower			: BYTE;										//% of the max Power in kW when the Device is manually on
	byPriority						: BYTE; 									//{#lynus.ag#()} //Priority of the device if controlled via the EMS block = 1 2 3 (If 0 then this device does not exist for the EMS block)
	byEnableSOC						: BYTE; 									//{#lynus.ag#()} //Enable the device when the battery SOC is greater than equal this value
	byDisableSOC					: BYTE; 									//{#lynus.ag#()} //Disable the device when the battery SOC is smaler than equal this value 
	rMaxPower						: REAL; 									//{#lynus.ag#()} //Max. power from the big consumer with unit kW
END_STRUCT
END_TYPE

// ---- Energy/DUTs/PV/ST_PV_Output.TcDUT
TYPE ST_PV_Output :
STRUCT
	bEnabled									: BOOL;									//Pv function is enabled
	byErrorWarning								: BYTE;									//Show if the function has a Error or a Warning
	lrTotalCounterEnergy_Consumption			: LREAL;								//Total Counter for Energy consumption with unit kWh
	lrTotalCounterEnergy_Production				: LREAL;								//Total Counter for Energy production with unit kWh
	lrCounterEnergyT1_Consumption				: LREAL;								//Total counter for energy Tariff 1 consumption with unit kWh
	lrCounterEnergyT2_Consumption				: LREAL;								//Total counter for energy Tariff 2 consumption with unit kWh
	lrCounterEnergyT1_Production				: LREAL;								//Total counter for energy Tariff 1 production with unit kWh
	lrCounterEnergyT2_Production				: LREAL;								//Total counter for energy Tariff 2 production with unit kWh
	lrPower										: LREAL;								//{#lynus.ag#()} //Pv power with unit kW
	lrPowerConsumption							: LREAL;								//Consumption pv with unit kW
	lrPowerProduction							: LREAL;								//Production pv with unit kW
	eMessage									: E_Message_PV;							//Message from the PV
END_STRUCT
END_TYPE

// ---- Energy/DUTs/Temperature/ST_InputData_KL320x.TcDUT
TYPE ST_InputData_KL320x :
STRUCT
	usiState			: USINT;					//Input State from KL320x
	iDataIn				: INT;						//Input Data from KL320x
END_STRUCT
END_TYPE

// ---- Energy/DUTs/Temperature/ST_OutputData_KL320x.TcDUT
TYPE ST_OutputData_KL320x :
STRUCT
	usiControl			: USINT;				//Output Control from KL320x
	iDataOut			: INT;					//Output Data from KL320x
END_STRUCT
END_TYPE

// ---- Energy/DUTs/Temperature/ST_Temperature_Output.TcDUT
TYPE ST_Temperature_Output :
STRUCT
	bEnabled						: BOOL;							//Temperature function is enabled
	rTemperature					: REAL;							//{#lynus.ag#()} //Temperature in °C
	byErrorWarning					: BYTE;							//Show if the function has a Error or a Warning
	eMessage						: E_Message_Temperature;		//Message from the Temperature
END_STRUCT
END_TYPE

// ---- Energy/DUTs/Valve Control/ST_Valve_Control_Output.TcDUT
TYPE ST_Valve_Control_Output :
STRUCT
	bEnabled						: BOOL;							//Valve control function is enabled
	bValvePos						: BOOL;							//{#lynus.ag#()} //Actual Valve Position
	byErrorWarning					: BYTE;							//Show if the function has a Error or a Warning
	eMessage						: E_Message_ValveControl;		//Message from the Valve position
END_STRUCT
END_TYPE

// ---- Energy/ENUMs Internal/Temperature/E_ChooseSensortype_KL320x.TcDUT
{attribute 'qualified_only'}
{attribute 'strict'}
{attribute 'conditionalshow'}
TYPE E_ChooseSensortype_KL320x :
(
	{attribute 'hide'}
	ePT100_KL320x := 0,							//Choose PT100 Measuring principle
	{attribute 'hide'}
	ePT1000_KL320x := 1,						//Choose PT1000 Measuring principle
	{attribute 'hide'}
	ePT10002Leiter_KL320x := 2,					//Choose PT1000 2-wire Measuring principle
	{attribute 'hide'}
	ePT500_KL320x := 3,							//Choose PT500 Measuring principle
	{attribute 'hide'}
	ePT200_KL320x := 4,							//Choose PT200 Measuring principle
	{attribute 'hide'}
	eNI100_KL320x := 5,							//Choose NI100 Measuring principle
	{attribute 'hide'}
	eNI1000_KL320x := 6,						//Choose NI1000 Measuring principle
	{attribute 'hide'}
	eNI120_KL320x := 7,							//Choose NI120 Measuring principle
	{attribute 'hide'}
	eResistor10Ohm5000Ohm_KL320x := 8,			//Selection resistance measurement 10 Ohm to 5000 Ohm
	{attribute 'hide'}
	eResistor10Ohm1200Ohm_KL320x := 9			//Selection resistance measurement 10 Ohm to 1200 Ohm
);
END_TYPE

// ---- Energy/ENUMs Internal/Temperature/E_Step_Config_Terminal_KL320x.TcDUT
{attribute 'qualified_only'}
{attribute 'strict'}
{attribute 'conditionalshow'}
TYPE E_Step_Config_Terminal_KL320x :
(
	{attribute 'hide'}
	eInit_KL320x := 0,													//Init Step terminal configuration
	{attribute 'hide'}
	eRegister31DeactivateWriteProtection_KL320x := 1,					//Register 31 deactivate write protection
	{attribute 'hide'}
	eChooseSensorType_KL320x := 2,										//Choose Sensor Type
	{attribute 'hide'}
	ePT100Config_KL320x := 3,											//Messurement principle PT100
	{attribute 'hide'}
	ePT1000Config_KL320x := 4,											//Messurement principle PT1000
	{attribute 'hide'}
	ePT10002WireConfig_KL320x := 5,										//Messurement principle PT1000 2 wire system
	{attribute 'hide'}
	ePT500Config_KL320x := 6,											//Messurement principle PT500
	{attribute 'hide'}
	ePT200Config_KL320x := 7,											//Messurement principle PT200
	{attribute 'hide'}
	eNI100Config_KL320x := 8,											//Messurement principle NI100
	{attribute 'hide'}
	eNI1000Config_KL320x := 9,											//Messurement principle NI1000
	{attribute 'hide'}
	eNI120Config_KL320x := 10,											//Messurement principle NI120
	{attribute 'hide'}
	e10Ohm5000OhmConfig_KL320x := 11,									//Resistor Messurement from 10Ohm to 5000Ohm
	{attribute 'hide'}
	e10Ohm1200OhmConfig_KL320x := 12,									//Resistor Messurement from 10Ohm to 1200Ohm
	{attribute 'hide'}
	eControlByteNull_KL320x := 13,										//Control Byte set to 0
	{attribute 'hide'}
	eRegister31ActivateWriteProtection_KL320x := 14,					//Register 31 activate write protection
	{attribute 'hide'}
	eReadConfiguration_KL320x := 15										//Read Configuration from terminal
);
END_TYPE

// ---- Energy/ENUMs/Battery Inverter/E_Message_BatteryInverter.TcDUT
{attribute 'qualified_only'}
{attribute 'strict'}
TYPE E_Message_BatteryInverter :
(
	eNoMessage := 0,
	eTooMuchBatteryInverter := 1,
	eBatteryInverterError := 2,
	eNoConnectionToBackend := 3
);
END_TYPE

// ---- Energy/ENUMs/Battery/E_Message_Battery.TcDUT
{attribute 'qualified_only'}
{attribute 'strict'}
TYPE E_Message_Battery :
(
	eNoMessage := 0,
	eTooMuchBattery := 1,
	eBatteryError := 2,
	eNoConnectionToBackend := 3
);
END_TYPE

// ---- Energy/ENUMs/Electric Charging Station/E_Message_ECS.TcDUT
{attribute 'qualified_only'}
{attribute 'strict'}
TYPE E_Message_ECS :
(
	eNoMessage := 0,
	eTooMuchECS := 1,
	eExternalLockActive := 2,
	eErrorECS := 3,
	eNoConnectionToBackend := 4,
	eWarningECS := 5
);
END_TYPE

// ---- Energy/ENUMs/Electric Heating Element/E_Message_EHE.TcDUT
{attribute 'qualified_only'}
{attribute 'strict'}
TYPE E_Message_EHE :
(
	eNoMessage := 0,
	eTooMuchEHE := 1,
	eLegionellaProtectionDisabledFromUser := 2,
	eTempSensorInBufferError := 3,
	eWindowsSystemTimeError := 4,
	eExternalLockActive := 5,
	eErrorEHE := 6,
	eEHEDontReachedTheSetTemp := 7,
	eNoConnectionToBackend := 8
);
END_TYPE

// ---- Energy/ENUMs/Electric Meter/E_Message_EM.TcDUT
{attribute 'qualified_only'}
{attribute 'strict'}
TYPE E_Message_EM :
(
	eNoMessage := 0,
	eTooMuchElectricMeter := 1,
	eElectricMeterError := 2,
	eNoConnectionToBackend := 3,
	eElectricMeterWarning :=4
);
END_TYPE

// ---- Energy/ENUMs/EMS/E_Message_EMS.TcDUT
{attribute 'qualified_only'}
{attribute 'strict'}
TYPE E_Message_EMS :
(
	eDisabled := 0,
	eEnabled := 1,
	eAllPrioritysAtMinimum := 2,
	eAllPrioritysAtMaximum := 3,
	eMissingPowerValuesOnDeviceSetup := 4,
	eTooMuchFunctionsInThisProject := 5,
	eNoConnectionToBackend := 6
);
END_TYPE

// ---- Energy/ENUMs/Generator/E_Message_Generator.TcDUT
{attribute 'qualified_only'}
{attribute 'strict'}
TYPE E_Message_Generator :
(
	eNoMessage := 0,
	eTooMuchGenerators := 1,
	eGeneratorError := 2,
	eNoConnectionToBackend := 3
);
END_TYPE

// ---- Energy/ENUMs/Grid/E_Message_Grid.TcDUT
{attribute 'qualified_only'}
{attribute 'strict'}
TYPE E_Message_Grid :
(
	eNoMessage := 0,
	eTooMuchGrids := 1,
	eGridError := 2,
	eNoConnectionToBackend := 3
);
END_TYPE

// ---- Energy/ENUMs/Heating Pump/E_Message_HP.TcDUT
{attribute 'qualified_only'}
{attribute 'strict'}
TYPE E_Message_HP :
(
	eNoMessage := 0,
	eTooMuchHP := 2,
	eExternalLockActive := 3,
	eExternalOnCommandIsActive := 4,
	eHPError := 5,
	eWindowsSystemTimeError := 6,
	eNoConnectionToBackend := 7,
	eConnectionError := 8
);
END_TYPE

// ---- Energy/ENUMs/House Consumption/E_Message_HouseC.TcDUT
{attribute 'qualified_only'}
{attribute 'strict'}
TYPE E_Message_HouseC :
(
	eNoMessage := 0,
	eTooMuchHouseC := 1,
	eErrorHouseC := 2,
	eNoConnectionToBackend := 3
);
END_TYPE

// ---- Energy/ENUMs/Other Big Consumer/E_Message_OBC.TcDUT
{attribute 'qualified_only'}
{attribute 'strict'}
TYPE E_Message_OBC :
(
	eNoMessage := 0,
	eTooMuchOBC := 2,
	eExternalLockActive := 3,
	eErrorOBC := 4,
	eNoConnectionToBackend := 5
);
END_TYPE

// ---- Energy/ENUMs/PV/E_Message_PV.TcDUT
{attribute 'qualified_only'}
{attribute 'strict'}
TYPE E_Message_PV :
(
	eNoMessage := 0,
	eTooMuchPV := 1,
	ePvError := 2,
	eNoConnectionToBackend := 3
);
END_TYPE

// ---- Energy/ENUMs/Temperature/E_Message_Temperature.TcDUT
{attribute 'qualified_only'}
{attribute 'strict'}
TYPE E_Message_Temperature :
(
	eNoMessage := 0,
	eTooMuchTemperature := 1,
	eTemperatureConfigError := 2,
	eTemperatureGeneralError := 3,
	eTemperatureOverrangeError := 4,
	eTemperatureUnderrangeError := 5,
	eNoConnectionToBackend := 6
);
END_TYPE

// ---- Energy/ENUMs/Valve Control/E_Message_ValveControl.TcDUT
{attribute 'qualified_only'}
{attribute 'strict'}
TYPE E_Message_ValveControl :
(
	eNoMessage := 0,
	eTooMuchValvePositions := 1,
	eValvePositionError := 2,
	eValvePositionIsControlledLocal := 3,
	eNoConnectionToBackend := 4,
	eTempSensorError := 5
);
END_TYPE

// ---- General/DUTs Internal/Convert/eByteOrder.TcDUT
{attribute 'qualified_only'}
{attribute 'strict'}
{attribute 'conditionalshow'}
TYPE eByteOrder :
(
	{attribute 'hide'}
	eBigEndian	:= 0,
	{attribute 'hide'}
	eLittleEndian	:= 1
);
END_TYPE

// ---- General/DUTs Internal/Convert/ST_UN_FLOAT_CONVERT_DWORD_REAL.TcDUT
{attribute 'conditionalshow'}
TYPE ST_UN_FLOAT_CONVERT_DWORD_REAL :
UNION
	{attribute 'hide'}
	dwRawValue				: DWORD;											//Raw value as dword
	{attribute 'hide'}
	rValueFloat				: REAL;												//Float value
END_UNION
END_TYPE

// ---- General/DUTs Internal/Convert/ST_UN_FLOAT_CONVERT_ULINT_LREAL.TcDUT
{attribute 'conditionalshow'}
TYPE ST_UN_FLOAT_CONVERT_ULINT_LREAL :
UNION
	{attribute 'hide'}
	uliRawValue				: ULINT;					//Raw value as ulint
	{attribute 'hide'}
	lrValueFloat			: LREAL;					//Float value
END_UNION
END_TYPE

// ---- General/DUTs Internal/Devices/ST_NumberOfDevices_GVL.TcDUT
{attribute 'conditionalshow'}
TYPE ST_NumberOfDevices_GVL :
STRUCT
	{attribute 'hide'}
	diNumberOfBatterys							: DINT;							//Number of Batterys on this plc project
	{attribute 'hide'}
	diNumberOfBatteryInverters					: DINT;							//Number of Battery Inverters on this plc project
	{attribute 'hide'}
	diNumberOfECS								: DINT;							//Number of Electric charging stations on this plc project
	{attribute 'hide'}
	diNumberOfEHE								: DINT;							//Number of Electric heating elements on this plc project
	{attribute 'hide'}
	diNumberOfElectricMeters					: DINT;							//Number of Electric meaters on this plc project
	{attribute 'hide'}
	diNumberOfGenerators						: DINT;							//Number of Generators on this plc project
	{attribute 'hide'}
	diNumberOfGrids								: DINT;							//Number of Grids on this plc project
	{attribute 'hide'}
	diNumberOfHP								: DINT;							//Number of Heating pumps on this plc project
	{attribute 'hide'}
	diNumberOfHouseConsumption					: DINT;							//Number of House consumption on this plc project
	{attribute 'hide'}
	diNumberOfOBC								: DINT;							//Number of other big consumer on this plc project
	{attribute 'hide'}
	diNumberOfPvSystems							: DINT;							//Number of Pv systems on this plc project
	{attribute 'hide'}
	diNumberOfEMS								: DINT;							//Number of EMS on this plc project
	{attribute 'hide'}
	diNumberOfValveControls						: DINT;							//Number of Valve Controls on this plc project
	{attribute 'hide'}
	diNumberOfSetPointOpt						: DINT;							//Number of Setpoint OPtimizer on this plc project
END_STRUCT
END_TYPE

// ---- Sensors/DUTs Internal/Temperature/ST_Temperature_GVL.TcDUT
{attribute 'conditionalshow'}
TYPE ST_Temperature_GVL :
STRUCT
	{attribute 'hide'}
	bEnabled						: BOOL;							//Temperature function is enabled
	{attribute 'hide'}
	rTemperature					: REAL;							//Temperature in °C
	{attribute 'hide'}
	byErrorWarning					: BYTE;							//Show if the function has a Error or a Warning
END_STRUCT
END_TYPE

// ---- GVL and CONST/Bussystems/Constants_Bussystems.TcGVL
{attribute 'qualified_only'}
{attribute 'conditionalshow'}
VAR_GLOBAL CONSTANT
	//Here we can set the limit for the RTU Master Functions
	{attribute 'hide'}
	diMaxNumberOfMBRTUMasterKL6xxx									: DINT := 15;
	//Here we can set the limit for the RTU Master Functions for the number of register
	{attribute 'hide'}
	wQuantityOfRegistersMBRTUMaster									: WORD := 250;
	//Here we can set the limit for the MBus Master Functions
	{attribute 'hide'}
	diMaxNumberOfMBusMasterKL6781									: DINT := 15;
	//Here we can set the limit for the KNX Master Functions
	{attribute 'hide'}
	diMaxNumberOfKNXMasterKL6301									: DINT := 15;
END_VAR

// ---- GVL and CONST/Bussystems/GVL_Bussystems.TcGVL
{attribute 'qualified_only'}
{attribute 'conditionalshow'}
VAR_GLOBAL		
	//Global Data from the RTU Masters
	{attribute 'hide'}
	stDataOfMBRTUMasterKL6xxx						: ARRAY[0..Constants_Bussystems.diMaxNumberOfMBRTUMasterKL6xxx]	OF ST_MBRTUMaster_KL6xxx_GVL;
	{attribute 'hide'}
	diNumberOfMBRTUMasters							: DINT;	//Number of RTU Masters on this plc project	
	//Global Data from the MBus Masters
	{attribute 'hide'}
	stDataOfMBusMasterKL6781						: ARRAY[0..Constants_Bussystems.diMaxNumberOfMBusMasterKL6781]	OF ST_MBusMaster_KL6781_GVL;
	{attribute 'hide'}
	diNumberOfMBusMasters							: DINT;	//Number of MBus Masters on this plc project
	//Global Data from the KNX Masters
	{attribute 'hide'}
	stDataOfKNXMasterKL6301							: ARRAY[0..Constants_Bussystems.diMaxNumberOfKNXMasterKL6301]	OF EIB_REC;
	{attribute 'hide'}
	diNumberOfKNXMasters							: DINT;	//Number of KNX Masters on this plc project
END_VAR

// ---- GVL and CONST/Energy/Constants_Energy.TcGVL
{attribute 'qualified_only'}
{attribute 'conditionalshow'}
VAR_GLOBAL CONSTANT
	//Here we can set the limits for the energy devices
	{attribute 'hide'}
	diMaxNumberOfBatterys												: DINT := 15;
	{attribute 'hide'}
	diMaxNumberOfBatteryInverters										: DINT := 15;
	{attribute 'hide'}
	diMaxNumberOfPvSystems												: DINT := 15;
	{attribute 'hide'}
	diMaxNumberOfGridConnections										: DINT := 15;
	{attribute 'hide'}
	diMaxNumberOfGenerators												: DINT := 15;
	{attribute 'hide'}
	diMaxNumberOfElectricHeatingElements								: DINT := 15;
	{attribute 'hide'}
	diMaxNumberOfHouseConsumptions										: DINT := 15;
	{attribute 'hide'}
	diMaxNumberOfHeatingPumps											: DINT := 15;
	{attribute 'hide'}	
	diMaxNumberOfElectricChargingStations								: DINT := 100;
	{attribute 'hide'}
	diMaxNumberOfOtherBigConsumers										: DINT := 30;
	{attribute 'hide'}
	diMaxNumberOfElectricMeters											: DINT := 150;
	{attribute 'hide'}
	diMaxNumberOfEMS													: DINT := 10;
	{attribute 'hide'}
	diMaxNumberOfValveControls											: DINT := 50;
	{attribute 'hide'}
	diMaxNumberOfSetPointOpt											: DINT := 50;
	//Target power limit in % to switch off the step switched and on/off devices
	{attribute 'hide'}
	byTargetOffPowerForOnOffDevices										: BYTE := 95;
	//Tolerance surplus/Consumption calculation EMS (Unit kW)
	{attribute 'hide'}
	rToleranceSurplusConsumption										: REAL := 0.05;
END_VAR

// ---- GVL and CONST/Energy/GVL_Energy.TcGVL
{attribute 'qualified_only'}
{attribute 'conditionalshow'}
VAR_GLOBAL
	//Global Data for all Energy Devices (The Array[0] or Array[0,0] must filled always with default values)
	{attribute 'hide'}
	stDataOfBatterys					: ARRAY[0..Constants_Energy.diMaxNumberOfEMS,0..Constants_Energy.diMaxNumberOfBatterys]						OF ST_Battery_GVL;	
	{attribute 'hide'}						
	stDataOfBatteryInverters			: ARRAY[0..Constants_Energy.diMaxNumberOfEMS,0..Constants_Energy.diMaxNumberOfBatteryInverters]				OF ST_BatteryInverter_GVL;
	{attribute 'hide'}		
	stDataGridConnections				: ARRAY[0..Constants_Energy.diMaxNumberOfEMS,0..Constants_Energy.diMaxNumberOfGridConnections]				OF ST_GridConnection_GVL;
	{attribute 'hide'}		
	stDataElectricHeatingElements		: ARRAY[0..Constants_Energy.diMaxNumberOfEMS,0..Constants_Energy.diMaxNumberOfElectricHeatingElements]		OF ST_EHE_GVL;	
	{attribute 'hide'}			
	stDataElectricChargingStations		: ARRAY[0..Constants_Energy.diMaxNumberOfEMS,0..Constants_Energy.diMaxNumberOfElectricChargingStations]		OF ST_ECS_GVL;
	{attribute 'hide'}					
	stDataHeatingPumps					: ARRAY[0..Constants_Energy.diMaxNumberOfEMS,0..Constants_Energy.diMaxNumberOfHeatingPumps] 				OF ST_HP_GVL;	
	{attribute 'hide'}				
	stDataOtherBigConsumers				: ARRAY[0..Constants_Energy.diMaxNumberOfEMS,0..Constants_Energy.diMaxNumberOfOtherBigConsumers]			OF ST_OBC_GVL;
	{attribute 'hide'}					
	stDataOfPvSystems					: ARRAY[0..Constants_Energy.diMaxNumberOfPvSystems]															OF ST_PV_GVL;
	{attribute 'hide'}
	stDataOfGenerators					: ARRAY[0..Constants_Energy.diMaxNumberOfGenerators]			 											OF ST_Generator_GVL;
	{attribute 'hide'}
	stDataHouseConsumptions				: ARRAY[0..Constants_Energy.diMaxNumberOfHouseConsumptions]													OF ST_HouseConsumption_GVL;
	{attribute 'hide'}
	stDataElectricMeters				: ARRAY[0..Constants_Energy.diMaxNumberOfElectricMeters]													OF ST_ElectricMeter_GVL;		
	{attribute 'hide'}
	stDataValveControls					: ARRAY[0..Constants_Energy.diMaxNumberOfValveControls]														OF ST_Valve_Control_GVL;		
	//Numbers from each Device on this plc
	{attribute 'hide'}
	stNumberOfDevices					: ST_NumberOfDevices_GVL;
END_VAR

// ---- GVL and CONST/Communicator/GVL_Communicator.TcGVL
{attribute 'qualified_only'}
{attribute 'conditionalshow'}
VAR_GLOBAL
	//Info Interface of al variable
	{attribute 'hide'}
	arrInterfaceInfoAlVariables				: ARRAY[1..10,1..Constants_Communicator.udiArraySizeMarkedSymobls] OF ST_Var_Info_GV;	//Info of all of found symbols in plc
	{attribute 'hide'}
	arrReadWriteArrayNumberInUse			: ARRAY[1..10] OF BOOL;																	//State from one array number if its just in use or not
	{attribute 'hide'}
	arrReadWriteArrayNumber					: ARRAY[1..10] OF BYTE;																	//Array Number Read Write
	{attribute 'hide'}
	arrCounterVariableInArray				: ARRAY[1..10] OF UDINT;																//Counter variables in output array
	{attribute 'hide'}
	bBusyInfoAlVariables					: BOOL;																					//Function Var Info Busy
	{attribute 'hide'}
	bErrorInfoAlVariables					: BOOL;																					//Function Var Info Error
	{attribute 'hide'}
	bInfoAlVariablesOK						: BOOL;																					//Necessary to start read/write and send/receive 
	{attribute 'hide'}
	byNumberOfReadWriteFunction				: BYTE;																					//Numbers of read write functions on plc
	//Value from read function <=> sending function and buffer
	{attribute 'hide'}
	arrInterfaceInfoValueSendTo				: ARRAY[1..10] OF ST_Var_Info_ValueSend_GV;												//read value and after that transport the data to the send function
	//Value from write function <=> received function and buffer
	{attribute 'hide'}
	arrInterfaceInfoValueWriteTo			: ARRAY[1..10] OF ST_Var_Info_ValueWrite_GV;											//write value on plc after received the data from the received function	
	//Indicates if we are connected with the Lynus Communicator to the Backend. (Withou this Lynus Functions not work after 7 Days)
	{attribute 'hide'}
	bStateConnectionToEnableFunctions		: BOOL;
END_VAR

// ---- GVL and CONST/Communicator/Constants_Communicator.TcGVL
{attribute 'qualified_only'}
{attribute 'conditionalshow'}
VAR_GLOBAL CONSTANT
	{attribute 'hide'}
	bySizeOfValueArray						: BYTE := 1;						//Size of the Array with the Values (Max 50)
	{attribute 'hide'}
	bySizeOfReceivedValueArrayInJson		: BYTE := 0;						//Size of the received Value Array from external in the json (Max 49) => bySizeOfReceivedValueArrayInJson = bySizeOfValueArray - 1 
	{attribute 'hide'}
	udiArraySizeSymbols						: UDINT := 1000;					//Size of the array from complete data of each one symbol in plc (Max 1000)
	{attribute 'hide'}
	udiArraySizeMarkedSymobls				: UDINT := 1500;					//Size of the array for all marked symbols incl. all Subitems (Max 2000) !!Change this for max variables!!
	{attribute 'hide'}
	uiArraySizeOfMarkedSubItems				: UINT := 100;						//Size of the array for marked Symbols in Subitems (Max 32768)
	{attribute 'hide'}
	uiArraySizeOfSubItems					: UINT := 200;						//Size of the array for all founded subitems after the Parse function(Max 1000)
END_VAR

// ---- GVL and CONST/General/Constants_General.TcGVL
{attribute 'qualified_only'}
{attribute 'conditionalshow'}
VAR_GLOBAL CONSTANT
	//Here we can set the time when all Lynus functions are dissabled without connection to the Lynus Backend
	{attribute 'hide'}
	tTimeDissableLynusFunctions							: TIME := T#11D;
END_VAR

// ---- GVL and CONST/Persistent Data/GVL_Persistent_Data.TcGVL
{attribute 'conditionalshow'}
VAR_GLOBAL
	{attribute 'hide'}
	bEventBasedActive			: BOOL;												//True, when the Event Based Mode is active
	{attribute 'hide'}
	bBusy						: BOOL;												//True, when the save procces is started
	{attribute 'hide'}
	bSaveData					: BOOL;												//Use to start to save the persistent data
	{attribute 'hide'}
	byNumberOfMasters			: BYTE;												//Number of Master FB's. Max 1 for each project on each plc
END_VAR

// ---- GVL and CONST/Sensors/Constants_Sensors.TcGVL
{attribute 'qualified_only'}
{attribute 'conditionalshow'}
VAR_GLOBAL CONSTANT
	//Here we can set the limits for the Sensor devices
	{attribute 'hide'}
	diMaxNumberOfTemperatureSensors										: DINT := 150;
	{attribute 'hide'}
	diMaxNumberOfKNXSensors												: DINT := 150;
END_VAR

// ---- GVL and CONST/Sensors/GVL_Sensors.TcGVL
{attribute 'qualified_only'}
{attribute 'conditionalshow'}
VAR_GLOBAL		
	//Global Data for all Temperatur Devices (The Array[0] or Array[0,0] must filled always with default values)
	{attribute 'hide'}
	stDataTemperatureSensors			: ARRAY[0..Constants_Sensors.diMaxNumberOfTemperatureSensors]				OF ST_Temperature_GVL;
	{attribute 'hide'}
	diNumberOfTemperatureSensors		: DINT; //Number of Temperature Sensors on this plc project		
	{attribute 'hide'}
	diNumberOfKNXSensors				: DINT; //Number of KNX Sensors on this plc project							
END_VAR

// ---- Bussystems/FBs Internal/KNX Master/FB_KNXMaster_Messages.TcPOU
{attribute 'conditionalshow'}
FUNCTION_BLOCK FB_KNXMaster_Messages
VAR_INPUT
	{attribute 'hide'}
	bErrorKNX							: BOOL;						//Error from the Mbus Function
	{attribute 'hide'}
	bErrorIntern						: BOOL;						//Internal Error
	{attribute 'hide'}
	bWarning							: BOOL;						//Warning from the RTU Function
	{attribute 'hide'}
	iWarningCode						: INT;						//Warning Code
	{attribute 'hide'}
	iErrorCode							: INT;						//Error Code		
END_VAR
VAR_OUTPUT
	{attribute 'hide'}
	byErrorWarning						: BYTE;						//Error Warning State
	eMessageKNXMaster					: E_Message_KNXMaster;		//Message from the KNX Master Function
END_VAR
VAR
END_VAR

//Creator : Kai Ebensperger
//Company : Lynus AG
//Date : 24.08.2021
//Version : 1.0.0.0

//With this Funciton is possible to handel the Error and Warning Codes from the KNX Master.

//Warnings
IF bWarning AND iWarningCode = 0 THEN
	eMessageKNXMaster := E_Message_KNXMaster.eNoConnectionToBackend;
END_IF

